C09199=1111.807,-65.980,-48.450,179.739,5.212,148.980
C09200=1111.812,-66.230,-48.440,179.738,5.207,148.979
C09201=1111.817,-66.480,-48.428,179.738,5.202,148.978
C09202=1111.823,-66.729,-48.417,179.737,5.197,148.977
C09203=1111.828,-66.979,-48.406,179.738,5.192,148.976
C09204=1111.833,-67.229,-48.395,179.737,5.187,148.975
C09205=1111.838,-67.478,-48.384,179.737,5.181,148.974
C09206=1111.843,-67.728,-48.373,179.737,5.176,148.972
C09207=1111.849,-67.978,-48.361,179.736,5.171,148.971
C09208=1111.854,-68.227,-48.350,179.737,5.166,148.970
C09209=1111.859,-68.477,-48.340,179.737,5.161,148.969
C09210=1111.864,-68.727,-48.328,179.736,5.155,148.968
C09211=1111.870,-68.976,-48.317,179.736,5.150,148.967
C09212=1111.875,-69.226,-48.306,179.736,5.145,148.966
C09213=1111.880,-69.475,-48.295,179.736,5.140,148.965
C09214=1111.885,-69.725,-48.285,179.736,5.135,148.964
C09215=1111.891,-69.975,-48.273,179.736,5.130,148.963
C09216=1111.896,-70.225,-48.263,179.735,5.124,148.962
C09217=1111.901,-70.475,-48.251,179.735,5.119,148.961
C09218=1111.906,-70.724,-48.240,179.735,5.114,148.959
C09219=1111.912,-70.974,-48.229,179.735,5.109,148.958
C09220=1111.917,-71.224,-48.218,179.735,5.104,148.957
C09221=1111.922,-71.473,-48.208,179.735,5.099,148.956
C09222=1111.927,-71.723,-48.197,179.735,5.094,148.955
C09223=1111.932,-71.972,-48.186,179.735,5.089,148.954
C09224=1111.937,-72.187,-48.176,179.735,5.084,148.953
C09225=1111.941,-72.403,-48.167,179.735,5.079,148.952
C09226=1111.946,-72.617,-48.157,179.735,5.075,148.951
C09227=1111.950,-72.832,-48.149,179.735,5.070,148.950
C09228=1111.955,-73.046,-48.139,179.735,5.066,148.949
C09229=1111.960,-73.262,-48.130,179.735,5.061,148.948
C09230=1111.963,-73.476,-48.120,179.735,5.057,148.947
C09231=1111.969,-73.691,-48.111,179.735,5.053,148.946
C09232=1111.973,-73.941,-48.100,179.735,5.048,148.945
C09233=1111.979,-74.190,-48.090,179.735,5.042,148.944
C09234=1111.984,-74.440,-48.079,179.735,5.037,148.943
C09235=1111.990,-74.690,-48.068,179.735,5.032,148.941
C09236=1111.995,-74.940,-48.057,179.736,5.027,148.940
C09237=1112.000,-75.189,-48.046,179.735,5.022,148.939
C09238=1112.005,-75.439,-48.036,179.735,5.017,148.938
C09239=1112.011,-75.689,-48.026,179.735,5.012,148.937
C09240=1112.016,-75.938,-48.014,179.736,5.007,148.936
C09241=1112.021,-76.188,-48.004,179.736,5.002,148.935
C09242=1112.026,-76.438,-47.993,179.735,4.996,148.933
C09243=1112.031,-76.687,-47.983,179.735,4.990,148.932
C09244=1112.037,-76.937,-47.971,179.736,4.985,148.931
C09245=1112.043,-77.187,-47.961,179.736,4.980,148.930
C09246=1112.048,-77.437,-47.950,179.736,4.975,148.929
C09247=1112.053,-77.686,-47.940,179.736,4.970,148.928
C09248=1112.058,-77.936,-47.929,179.736,4.965,148.926
C09249=1112.064,-78.186,-47.919,179.736,4.960,148.925
C09250=1112.068,-78.436,-47.908,179.737,4.954,148.924
C09251=1112.074,-78.685,-47.897,179.737,4.949,148.923
C09252=1112.079,-78.935,-47.887,179.737,4.944,148.922
C09253=1112.085,-79.185,-47.877,179.737,4.939,148.921
C09254=1112.089,-79.435,-47.865,179.737,4.934,148.919
C09255=1112.095,-79.684,-47.855,179.737,4.929,148.918
C09256=1112.100,-79.934,-47.845,179.738,4.924,148.917
C09257=1112.105,-80.184,-47.834,179.738,4.918,148.916
C09258=1112.111,-80.433,-47.823,179.738,4.914,148.915
C09259=1112.116,-80.683,-47.813,179.739,4.909,148.914
C09260=1112.121,-80.933,-47.803,179.739,4.903,148.912
C09261=1112.126,-81.183,-47.792,179.739,4.898,148.911
C09262=1112.132,-81.432,-47.782,179.740,4.893,148.910
C09263=1112.137,-81.683,-47.771,179.740,4.888,148.909
C09264=1112.142,-81.932,-47.760,179.740,4.883,148.907
C09265=1112.148,-82.181,-47.750,179.740,4.878,148.906
C09266=1112.153,-82.431,-47.740,179.740,4.873,148.905
C09267=1112.158,-82.681,-47.729,179.740,4.867,148.904
C09268=1112.163,-82.931,-47.719,179.741,4.862,148.903
C09269=1112.169,-83.181,-47.709,179.741,4.857,148.902
C09270=1112.174,-83.430,-47.699,179.742,4.853,148.900
C09271=1112.179,-83.680,-47.688,179.742,4.847,148.899
C09272=1112.184,-83.929,-47.677,179.742,4.842,148.898
C09273=1112.189,-84.179,-47.667,179.743,4.837,148.897
C09274=1112.195,-84.429,-47.657,179.743,4.832,148.895
C09275=1112.200,-84.678,-47.646,179.743,4.827,148.894
C09276=1112.205,-84.929,-47.636,179.744,4.822,148.893
C09277=1112.211,-85.178,-47.626,179.744,4.817,148.892
C09278=1112.216,-85.428,-47.615,179.744,4.812,148.891
C09279=1112.221,-85.678,-47.605,179.745,4.806,148.889
C09280=1112.226,-85.892,-47.597,179.745,4.802,148.888
C09281=1112.230,-86.108,-47.588,179.745,4.799,148.887
C09282=1112.235,-86.322,-47.579,179.745,4.793,148.886
C09283=1112.239,-86.538,-47.570,179.746,4.789,148.885
C09284=1112.244,-86.752,-47.561,179.746,4.785,148.884
C09285=1112.248,-86.967,-47.552,179.747,4.781,148.883
C09286=1112.253,-87.182,-47.543,179.746,4.776,148.882
C09287=1112.257,-87.397,-47.534,179.747,4.772,148.881
C09288=1112.263,-87.646,-47.524,179.747,4.767,148.880
C09289=1112.268,-87.896,-47.514,179.748,4.763,148.879
C09290=1112.273,-88.146,-47.504,179.748,4.757,148.877
C09291=1112.278,-88.395,-47.494,179.748,4.752,148.876
C09292=1112.284,-88.645,-47.483,179.749,4.747,148.875
C09293=1112.289,-88.896,-47.474,179.750,4.742,148.874
C09294=1112.295,-89.145,-47.463,179.750,4.737,148.872
C09295=1112.300,-89.395,-47.454,179.750,4.732,148.871
C09296=1112.305,-89.644,-47.444,179.751,4.728,148.870
C09297=1112.310,-89.894,-47.433,179.751,4.723,148.869
C09298=1112.316,-90.144,-47.423,179.751,4.717,148.868
C09299=1112.321,-90.393,-47.413,179.753,4.713,148.866
C09300=1112.326,-90.643,-47.403,179.753,4.707,148.865
C09301=1112.331,-90.893,-47.392,179.753,4.702,148.864
C09302=1112.337,-91.143,-47.382,179.754,4.698,148.863
C09303=1112.341,-91.392,-47.372,179.754,4.693,148.862
C09304=1112.347,-91.643,-47.363,179.754,4.688,148.860
C09305=1112.353,-91.892,-47.353,179.755,4.683,148.859
C09306=1112.358,-92.142,-47.342,179.755,4.678,148.858
C09307=1112.362,-92.392,-47.332,179.757,4.673,148.857
C09308=1112.368,-92.641,-47.322,179.757,4.668,148.855
C09309=1112.374,-92.891,-47.312,179.758,4.664,148.854
C09310=1112.380,-93.141,-47.302,179.758,4.659,148.853
C09311=1112.384,-93.391,-47.292,179.758,4.654,148.852
C09312=1112.389,-93.640,-47.282,179.759,4.649,148.851
C09313=1112.395,-93.890,-47.272,179.759,4.644,148.849
C09314=1112.400,-94.139,-47.262,179.760,4.640,148.848
C09315=1112.405,-94.390,-47.253,179.760,4.635,148.847
C09316=1112.411,-94.640,-47.242,179.760,4.630,148.846
C09317=1112.416,-94.889,-47.233,179.761,4.625,148.845
C09318=1112.421,-95.138,-47.223,179.761,4.620,148.843
C09319=1112.426,-95.389,-47.212,179.761,4.615,148.842
C09320=1112.431,-95.638,-47.203,179.762,4.611,148.841
C09321=1112.437,-95.888,-47.193,179.762,4.605,148.840
C09322=1112.443,-96.138,-47.183,179.763,4.600,148.839
C09323=1112.448,-96.387,-47.174,179.763,4.595,148.838
C09324=1112.453,-96.638,-47.163,179.764,4.591,148.836
C09325=1112.458,-96.887,-47.153,179.764,4.586,148.835
C09326=1112.463,-97.136,-47.143,179.764,4.580,148.834
C09327=1112.469,-97.387,-47.134,179.765,4.576,148.833
C09328=1112.475,-97.636,-47.124,179.765,4.571,148.832
C09329=1112.479,-97.886,-47.114,179.765,4.566,148.830
C09330=1112.485,-98.136,-47.104,179.765,4.561,148.829
C09331=1112.490,-98.385,-47.095,179.766,4.556,148.828
C09332=1112.495,-98.635,-47.084,179.766,4.551,148.827
C09333=1112.501,-98.885,-47.075,179.767,4.546,148.826
C09334=1112.506,-99.134,-47.065,179.767,4.541,148.824
C09335=1112.511,-99.385,-47.055,179.768,4.536,148.823
C09336=1112.516,-99.600,-47.047,179.767,4.532,148.822
C09337=1112.520,-99.814,-47.039,179.768,4.528,148.821
C09338=1112.524,-100.029,-47.030,179.769,4.523,148.820
C09339=1112.530,-100.245,-47.022,179.769,4.519,148.819
C09340=1112.534,-100.459,-47.013,179.769,4.515,148.818
C09341=1112.538,-100.674,-47.005,179.769,4.510,148.817
C09342=1112.543,-100.889,-46.996,179.770,4.506,148.816
C09343=1112.548,-101.104,-46.988,179.770,4.502,148.815
C09344=1112.553,-101.353,-46.979,179.770,4.497,148.814
C09345=1112.559,-101.604,-46.969,179.770,4.492,148.813
C09346=1112.563,-101.854,-46.959,179.771,4.487,148.812
C09347=1112.569,-102.103,-46.949,179.771,4.483,148.810
C09348=1112.574,-102.353,-46.940,179.772,4.477,148.809
C09349=1112.580,-102.603,-46.930,179.772,4.472,148.808
C09350=1112.585,-102.852,-46.921,179.772,4.467,148.807
C09351=1112.590,-103.102,-46.911,179.772,4.462,148.806
C09352=1112.596,-103.352,-46.902,179.773,4.458,148.804
C09353=1112.601,-103.601,-46.892,179.773,4.452,148.803
C09354=1112.606,-103.852,-46.882,179.774,4.447,148.802
C09355=1112.611,-104.101,-46.872,179.774,4.442,148.801
C09356=1112.617,-104.336,-46.864,179.775,4.438,148.800
C09357=1112.621,-104.571,-46.854,179.774,4.433,148.799
C09358=1112.626,-104.806,-46.846,179.775,4.428,148.797
C09359=1112.631,-105.041,-46.837,179.775,4.423,148.796
C09360=1112.637,-105.276,-46.828,179.776,4.418,148.795
C09361=1112.641,-105.511,-46.818,179.776,4.414,148.794
C09362=1112.646,-105.746,-46.810,179.776,4.409,148.793
C09363=1112.651,-105.980,-46.801,179.776,4.404,148.792
C09364=1112.656,-106.230,-46.792,179.777,4.400,148.790
C09365=1112.662,-106.480,-46.782,179.777,4.395,148.789
C09366=1112.667,-106.730,-46.773,179.778,4.389,148.788
C09367=1112.673,-106.980,-46.763,179.778,4.384,148.787
C09368=1112.678,-107.229,-46.754,179.778,4.379,148.786
C09369=1112.683,-107.479,-46.744,179.778,4.374,148.784
C09370=1112.689,-107.729,-46.735,179.779,4.370,148.783
C09371=1112.693,-107.978,-46.726,179.780,4.364,148.782
C09372=1112.699,-108.228,-46.716,179.780,4.359,148.781
C09373=1112.704,-108.478,-46.706,179.780,4.354,148.780
C09374=1112.709,-108.728,-46.698,179.780,4.349,148.778
C09375=1112.715,-108.978,-46.688,179.781,4.344,148.777
C09376=1112.720,-109.227,-46.678,179.781,4.339,148.776
C09377=1112.726,-109.477,-46.669,179.782,4.334,148.775
C09378=1112.731,-109.727,-46.660,179.782,4.329,148.774
C09379=1112.736,-109.976,-46.650,179.782,4.324,148.772
C09380=1112.742,-110.226,-46.641,179.782,4.319,148.771
C09381=1112.747,-110.476,-46.632,179.783,4.313,148.770
C09382=1112.752,-110.725,-46.622,179.783,4.308,148.769
C09383=1112.758,-110.976,-46.613,179.784,4.303,148.767
C09384=1112.763,-111.225,-46.604,179.784,4.298,148.766
C09385=1112.768,-111.475,-46.595,179.784,4.293,148.765
C09386=1112.774,-111.725,-46.585,179.785,4.288,148.764
C09387=1112.779,-111.975,-46.576,179.785,4.283,148.763
C09388=1112.784,-112.225,-46.567,179.785,4.278,148.761
C09389=1112.789,-112.474,-46.558,179.786,4.273,148.760
C09390=1112.795,-112.724,-46.548,179.786,4.268,148.759
C09391=1112.800,-112.974,-46.539,179.786,4.262,148.758
C09392=1112.805,-113.204,-46.531,179.787,4.257,148.757
C09393=1112.810,-113.434,-46.523,179.787,4.253,148.755
C09394=1112.815,-113.663,-46.514,179.788,4.248,148.754
C09395=1112.820,-113.893,-46.505,179.787,4.243,148.753
C09396=1112.825,-114.124,-46.497,179.788,4.239,148.752
C09397=1112.829,-114.354,-46.489,179.788,4.233,148.751
C09398=1112.834,-114.584,-46.480,179.789,4.229,148.750
C09399=1112.840,-114.813,-46.472,179.789,4.224,148.749
C09400=1112.845,-115.063,-46.463,179.789,4.219,148.747
C09401=1112.850,-115.313,-46.454,179.790,4.214,148.746
C09402=1112.856,-115.563,-46.444,179.790,4.208,148.745
C09403=1112.861,-115.812,-46.435,179.791,4.203,148.743
C09404=1112.866,-116.062,-46.426,179.791,4.198,148.742
C09405=1112.871,-116.312,-46.417,179.791,4.193,148.741
C09406=1112.876,-116.562,-46.408,179.791,4.188,148.740
C09407=1112.882,-116.812,-46.399,179.792,4.183,148.739
C09408=1112.888,-117.061,-46.390,179.792,4.177,148.737
C09409=1112.893,-117.311,-46.381,179.793,4.172,148.736
C09410=1112.898,-117.561,-46.372,179.793,4.167,148.735
C09411=1112.903,-117.810,-46.363,179.793,4.162,148.734
C09412=1112.909,-118.061,-46.354,179.794,4.156,148.732
C09413=1112.915,-118.310,-46.345,179.794,4.151,148.731
C09414=1112.919,-118.560,-46.335,179.795,4.146,148.730
C09415=1112.925,-118.810,-46.327,179.795,4.141,148.728
C09416=1112.930,-119.059,-46.318,179.795,4.135,148.727
C09417=1112.935,-119.309,-46.309,179.796,4.130,148.726
C09418=1112.941,-119.558,-46.300,179.796,4.125,148.725
C09419=1112.947,-119.809,-46.291,179.797,4.119,148.723
C09420=1112.952,-120.058,-46.282,179.797,4.114,148.722
C09421=1112.957,-120.308,-46.273,179.797,4.109,148.721
C09422=1112.962,-120.558,-46.264,179.797,4.104,148.720
C09423=1112.968,-120.807,-46.255,179.798,4.098,148.718
C09424=1112.973,-121.057,-46.247,179.799,4.093,148.717
C09425=1112.978,-121.307,-46.238,179.799,4.088,148.716
C09426=1112.984,-121.557,-46.229,179.799,4.083,148.715
C09427=1112.989,-121.807,-46.221,179.800,4.077,148.713
C09428=1112.994,-122.057,-46.212,179.800,4.072,148.712
C09429=1113.000,-122.306,-46.203,179.800,4.066,148.711
C09430=1113.006,-122.556,-46.194,179.800,4.061,148.710
C09431=1113.011,-122.806,-46.185,179.801,4.056,148.708
C09432=1113.016,-123.056,-46.176,179.801,4.050,148.707
C09433=1113.021,-123.306,-46.167,179.802,4.045,148.706
C09434=1113.027,-123.555,-46.158,179.802,4.040,148.704
C09435=1113.032,-123.805,-46.150,179.803,4.034,148.703
C09436=1113.037,-124.055,-46.141,179.803,4.029,148.702
C09437=1113.043,-124.305,-46.132,179.804,4.024,148.700
C09438=1113.048,-124.555,-46.124,179.804,4.019,148.699
C09439=1113.054,-124.804,-46.115,179.804,4.013,148.698
C09440=1113.059,-125.054,-46.106,179.805,4.007,148.696
C09441=1113.064,-125.304,-46.097,179.805,4.002,148.695
C09442=1113.069,-125.554,-46.088,179.805,3.997,148.694
C09443=1113.075,-125.804,-46.081,179.806,3.991,148.692
C09444=1113.080,-126.054,-46.072,179.806,3.986,148.691
C09445=1113.086,-126.303,-46.063,179.807,3.981,148.690
C09446=1113.091,-126.553,-46.054,179.807,3.974,148.689
C09447=1113.096,-126.802,-46.045,179.807,3.969,148.687
C09448=1113.101,-127.018,-46.039,179.808,3.965,148.686
C09449=1113.105,-127.234,-46.031,179.808,3.960,148.685
C09450=1113.110,-127.449,-46.023,179.808,3.955,148.684
C09451=1113.115,-127.664,-46.016,179.809,3.951,148.683
C09452=1113.119,-127.879,-46.009,179.809,3.946,148.682
C09453=1113.124,-128.094,-46.001,179.810,3.942,148.681
C09454=1113.128,-128.309,-45.994,179.810,3.936,148.679
C09455=1113.132,-128.523,-45.987,179.810,3.932,148.678
C09456=1112.710,-128.514,-46.013,179.818,3.936,148.677
C09457=1112.703,-128.193,-46.024,179.817,3.943,148.679
C09458=1112.697,-127.871,-46.035,179.817,3.950,148.680
C09459=1112.690,-127.549,-46.046,179.816,3.957,148.682
C09460=1112.683,-127.227,-46.057,179.816,3.964,148.684
C09461=1112.677,-126.978,-46.065,179.815,3.970,148.685
C09462=1112.671,-126.728,-46.074,179.814,3.975,148.686
C09463=1112.666,-126.478,-46.083,179.814,3.980,148.688
C09464=1112.661,-126.228,-46.092,179.813,3.986,148.689
C09465=1112.655,-125.979,-46.100,179.813,3.991,148.690
C09466=1112.650,-125.728,-46.109,179.813,3.997,148.691
C09467=1112.645,-125.479,-46.118,179.812,4.003,148.693
C09468=1112.639,-125.229,-46.126,179.812,4.008,148.694
C09469=1112.634,-124.980,-46.135,179.811,4.013,148.696
C09470=1112.629,-124.730,-46.144,179.811,4.018,148.697
C09471=1112.623,-124.480,-46.153,179.811,4.024,148.698
C09472=1112.618,-124.230,-46.162,179.810,4.029,148.700
C09473=1112.613,-123.980,-46.171,179.810,4.034,148.701
C09474=1112.607,-123.730,-46.178,179.810,4.040,148.702
C09475=1112.602,-123.481,-46.187,179.809,4.046,148.703
C09476=1112.597,-123.231,-46.196,179.809,4.051,148.705
C09477=1112.591,-122.981,-46.205,179.809,4.056,148.706
C09478=1112.586,-122.731,-46.214,179.808,4.061,148.707
C09479=1112.581,-122.481,-46.223,179.807,4.067,148.709
C09480=1112.575,-122.232,-46.231,179.807,4.072,148.710
C09481=1112.570,-121.982,-46.240,179.807,4.077,148.711
C09482=1112.565,-121.732,-46.249,179.806,4.083,148.712
C09483=1112.560,-121.482,-46.258,179.806,4.088,148.714
C09484=1112.554,-121.232,-46.268,179.805,4.093,148.715
C09485=1112.549,-120.982,-46.277,179.805,4.098,148.716
C09486=1112.543,-120.733,-46.285,179.804,4.104,148.718
C09487=1112.538,-120.483,-46.294,179.804,4.109,148.719
C09488=1112.533,-120.234,-46.303,179.804,4.114,148.720
C09489=1112.527,-119.984,-46.312,179.804,4.119,148.721
C09490=1112.522,-119.734,-46.321,179.803,4.126,148.723
C09491=1112.517,-119.484,-46.330,179.803,4.131,148.724
C09492=1112.511,-119.234,-46.339,179.803,4.136,148.725
C09493=1112.505,-118.985,-46.348,179.802,4.141,148.726
C09494=1112.500,-118.735,-46.356,179.802,4.146,148.727
C09495=1112.495,-118.485,-46.365,179.801,4.152,148.729
C09496=1112.490,-118.235,-46.374,179.801,4.157,148.730
C09497=1112.485,-117.985,-46.383,179.801,4.162,148.731
C09498=1112.479,-117.735,-46.393,179.801,4.167,148.733
C09499=1112.474,-117.486,-46.402,179.800,4.173,148.734
C09500=1112.469,-117.236,-46.411,179.800,4.178,148.735
C09501=1112.464,-116.986,-46.420,179.799,4.183,148.736
C09502=1112.458,-116.737,-46.429,179.799,4.188,148.738
C09503=1112.452,-116.487,-46.438,179.799,4.194,148.739
C09504=1112.447,-116.237,-46.447,179.798,4.198,148.740
C09505=1112.442,-115.987,-46.456,179.798,4.203,148.741
C09506=1112.437,-115.737,-46.465,179.797,4.209,148.743
C09507=1112.431,-115.488,-46.475,179.797,4.214,148.744
C09508=1112.426,-115.238,-46.484,179.796,4.219,148.745
C09509=1112.421,-115.020,-46.492,179.797,4.224,148.746
C09510=1112.417,-114.804,-46.499,179.796,4.228,148.747
C09511=1112.412,-114.589,-46.507,179.796,4.233,148.748
C09512=1112.408,-114.374,-46.516,179.795,4.237,148.749
C09513=1112.403,-114.159,-46.523,179.795,4.241,148.750
C09514=1112.398,-113.944,-46.531,179.795,4.246,148.751
C09515=1112.394,-113.729,-46.539,179.794,4.250,148.753
C09516=1112.389,-113.514,-46.547,179.794,4.255,148.754
C09517=1112.384,-113.299,-46.554,179.794,4.259,148.755
C09518=1112.380,-113.084,-46.563,179.793,4.263,148.756
C09519=1112.375,-112.834,-46.572,179.793,4.269,148.757
C09520=1112.369,-112.584,-46.582,179.793,4.274,148.758
C09521=1112.364,-112.334,-46.590,179.792,4.279,148.759
C09522=1112.359,-112.085,-46.600,179.792,4.284,148.761
C09523=1112.353,-111.834,-46.610,179.791,4.290,148.762
C09524=1112.348,-111.585,-46.618,179.791,4.295,148.763
C09525=1112.343,-111.335,-46.628,179.791,4.300,148.764
C09526=1112.337,-111.085,-46.638,179.791,4.305,148.766
C09527=1112.332,-110.835,-46.646,179.790,4.309,148.767
C09528=1112.327,-110.586,-46.656,179.790,4.315,148.768
C09529=1112.321,-110.336,-46.666,179.789,4.320,148.769
C09530=1112.316,-110.086,-46.674,179.789,4.325,148.770
C09531=1112.311,-109.837,-46.684,179.789,4.330,148.772
C09532=1112.305,-109.587,-46.694,179.789,4.335,148.773
C09533=1112.300,-109.337,-46.702,179.788,4.340,148.774
C09534=1112.295,-109.087,-46.713,179.788,4.346,148.775
C09535=1112.289,-108.837,-46.722,179.787,4.350,148.776
C09536=1112.284,-108.588,-46.730,179.787,4.355,148.778
C09537=1112.279,-108.338,-46.741,179.786,4.361,148.779
C09538=1112.274,-108.088,-46.750,179.786,4.366,148.780
C09539=1112.268,-107.839,-46.760,179.786,4.371,148.782
C09540=1112.263,-107.589,-46.769,179.786,4.376,148.783
C09541=1112.258,-107.339,-46.778,179.785,4.381,148.784
C09542=1112.252,-107.089,-46.788,179.784,4.386,148.785
C09543=1112.247,-106.840,-46.797,179.784,4.391,148.786
C09544=1112.241,-106.590,-46.807,179.784,4.396,148.788
C09545=1112.236,-106.340,-46.816,179.784,4.401,148.789
C09546=1112.231,-106.091,-46.825,179.784,4.406,148.790
C09547=1112.226,-105.840,-46.835,179.783,4.411,148.791
C09548=1112.221,-105.590,-46.844,179.782,4.416,148.792
C09549=1112.215,-105.341,-46.854,179.782,4.421,148.794
C09550=1112.210,-105.091,-46.863,179.782,4.426,148.795
C09551=1112.204,-104.841,-46.873,179.782,4.431,148.796
C09552=1112.199,-104.591,-46.882,179.782,4.436,148.797
C09553=1112.194,-104.342,-46.893,179.781,4.441,148.798
C09554=1112.188,-104.092,-46.901,179.780,4.446,148.800
C09555=1112.183,-103.843,-46.912,179.780,4.451,148.801
C09556=1112.178,-103.593,-46.921,179.780,4.456,148.802
C09557=1112.173,-103.342,-46.931,179.780,4.461,148.803
C09558=1112.168,-103.093,-46.941,179.779,4.466,148.804
C09559=1112.162,-102.843,-46.950,179.779,4.471,148.806
C09560=1112.157,-102.594,-46.960,179.778,4.476,148.807
C09561=1112.151,-102.344,-46.969,179.778,4.481,148.808
C09562=1112.146,-102.094,-46.979,179.778,4.486,148.809
C09563=1112.140,-101.844,-46.988,179.777,4.491,148.810
C09564=1112.136,-101.594,-46.998,179.777,4.496,148.812
C09565=1112.131,-101.345,-47.009,179.777,4.501,148.813
C09566=1112.125,-101.095,-47.018,179.777,4.506,148.814
C09567=1112.120,-100.880,-47.026,179.776,4.510,148.815
C09568=1112.116,-100.666,-47.035,179.775,4.514,148.816
C09569=1112.111,-100.450,-47.043,179.775,4.518,148.817
C09570=1112.107,-100.235,-47.051,179.775,4.523,148.818
C09571=1112.102,-100.021,-47.060,179.775,4.527,148.819
C09572=1112.098,-99.805,-47.069,179.774,4.531,148.820
C09573=1112.093,-99.590,-47.076,179.774,4.535,148.821
C09574=1112.088,-99.376,-47.085,179.774,4.540,148.822
C09575=1112.083,-99.126,-47.095,179.774,4.545,148.823
C09576=1112.079,-98.876,-47.105,179.773,4.550,148.824
C09577=1112.073,-98.626,-47.114,179.773,4.555,148.826
C09578=1112.067,-98.377,-47.125,179.773,4.560,148.827
C09579=1112.062,-98.127,-47.134,179.772,4.564,148.828
C09580=1112.057,-97.877,-47.144,179.772,4.570,148.829
C09581=1112.051,-97.627,-47.154,179.772,4.575,148.830
C09582=1112.046,-97.378,-47.164,179.771,4.579,148.832
C09583=1112.041,-97.128,-47.173,179.771,4.584,148.833
C09584=1112.035,-96.878,-47.184,179.770,4.589,148.834
C09585=1112.031,-96.628,-47.194,179.770,4.594,148.835
C09586=1112.025,-96.379,-47.204,179.769,4.599,148.836
C09587=1112.019,-96.128,-47.213,179.769,4.604,148.838
C09588=1112.014,-95.879,-47.223,179.769,4.609,148.839
C09589=1112.009,-95.630,-47.233,179.769,4.614,148.840
C09590=1112.004,-95.379,-47.244,179.768,4.619,148.841
C09591=1111.999,-95.130,-47.253,179.768,4.624,148.842
C09592=1111.993,-94.880,-47.263,179.768,4.629,148.843
C09593=1111.987,-94.631,-47.273,179.767,4.633,148.845
C09594=1111.983,-94.381,-47.283,179.767,4.638,148.846
C09595=1111.978,-94.131,-47.293,179.766,4.644,148.847
C09596=1111.972,-93.882,-47.303,179.766,4.648,148.848
C09597=1111.967,-93.632,-47.312,179.765,4.653,148.849
C09598=1111.962,-93.381,-47.323,179.765,4.657,148.851
C09599=1111.956,-93.132,-47.333,179.764,4.663,148.852
C09600=1111.951,-92.882,-47.343,179.764,4.667,148.853
C09601=1111.946,-92.632,-47.353,179.763,4.672,148.854
C09602=1111.941,-92.383,-47.363,179.763,4.678,148.856
C09603=1111.935,-92.133,-47.373,179.762,4.682,148.857
C09604=1111.929,-91.883,-47.383,179.762,4.687,148.858
C09605=1111.925,-91.633,-47.393,179.761,4.691,148.859
C09606=1111.919,-91.384,-47.403,179.761,4.697,148.860
C09607=1111.914,-91.134,-47.414,179.761,4.702,148.862
C09608=1111.909,-90.884,-47.424,179.760,4.706,148.863
C09609=1111.904,-90.635,-47.434,179.760,4.711,148.864
C09610=1111.898,-90.385,-47.444,179.759,4.717,148.865
C09611=1111.893,-90.136,-47.454,179.758,4.721,148.867
C09612=1111.888,-89.885,-47.465,179.758,4.726,148.868
C09613=1111.882,-89.636,-47.475,179.758,4.731,148.869
C09614=1111.877,-89.387,-47.485,179.757,4.736,148.870
C09615=1111.872,-89.136,-47.494,179.757,4.741,148.871
C09616=1111.866,-88.886,-47.505,179.757,4.746,148.872
C09617=1111.861,-88.637,-47.515,179.755,4.751,148.874
C09618=1111.856,-88.386,-47.525,179.755,4.756,148.875
C09619=1111.851,-88.137,-47.535,179.755,4.761,148.876
C09620=1111.845,-87.888,-47.545,179.755,4.766,148.877
C09621=1111.840,-87.637,-47.556,179.754,4.771,148.879
C09622=1111.835,-87.388,-47.566,179.754,4.776,148.880
C09623=1111.831,-87.173,-47.575,179.753,4.780,148.881
C09624=1111.826,-86.958,-47.584,179.753,4.785,148.882
C09625=1111.821,-86.744,-47.593,179.753,4.789,148.883
C09626=1111.817,-86.528,-47.602,179.752,4.793,148.884
C09627=1111.812,-86.314,-47.610,179.752,4.797,148.885
C09628=1111.808,-86.099,-47.620,179.752,4.802,148.886
C09629=1111.803,-85.884,-47.628,179.752,4.806,148.887
C09630=1111.799,-85.669,-47.637,179.751,4.811,148.888
C09631=1111.794,-85.419,-47.647,179.751,4.816,148.889
C09632=1111.789,-85.169,-47.657,179.750,4.821,148.891
C09633=1111.783,-84.920,-47.668,179.750,4.826,148.892
C09634=1111.778,-84.671,-47.678,179.750,4.830,148.893
C09635=1111.773,-84.420,-47.689,179.749,4.836,148.894
C09636=1111.767,-84.171,-47.699,179.749,4.841,148.895
C09637=1111.761,-83.921,-47.709,179.749,4.846,148.897
C09638=1111.756,-83.671,-47.720,179.748,4.851,148.898
C09639=1111.751,-83.422,-47.730,179.748,4.856,148.899
C09640=1111.746,-83.171,-47.741,179.748,4.862,148.900
C09641=1111.741,-82.922,-47.750,179.747,4.866,148.901
C09642=1111.736,-82.672,-47.762,179.747,4.871,148.903
C09643=1111.731,-82.423,-47.772,179.747,4.876,148.904
C09644=1111.725,-82.173,-47.782,179.747,4.881,148.905
C09645=1111.720,-81.923,-47.793,179.747,4.887,148.906
C09646=1111.715,-81.674,-47.803,179.746,4.892,148.907
C09647=1111.710,-81.424,-47.814,179.746,4.897,148.909
C09648=1111.704,-81.174,-47.824,179.746,4.902,148.910
C09649=1111.699,-80.924,-47.835,179.745,4.908,148.911
C09650=1111.694,-80.675,-47.845,179.745,4.913,148.912
C09651=1111.688,-80.425,-47.855,179.745,4.918,148.913
C09652=1111.683,-80.175,-47.867,179.745,4.923,148.915
C09653=1111.678,-79.926,-47.877,179.745,4.928,148.916
C09654=1111.673,-79.676,-47.888,179.745,4.933,148.917
C09655=1111.667,-79.426,-47.898,179.744,4.938,148.918
C09656=1111.662,-79.176,-47.909,179.744,4.943,148.919
C09657=1111.657,-78.927,-47.919,179.744,4.948,148.921
C09658=1111.652,-78.677,-47.930,179.743,4.953,148.922
C09659=1111.646,-78.427,-47.940,179.743,4.958,148.923
C09660=1111.641,-78.177,-47.952,179.743,4.963,148.924
C09661=1111.635,-77.928,-47.962,179.743,4.968,148.925
C09662=1111.630,-77.677,-47.973,179.743,4.974,148.926
C09663=1111.625,-77.428,-47.984,179.743,4.979,148.928
C09664=1111.620,-77.178,-47.994,179.742,4.984,148.929
C09665=1111.614,-76.929,-48.004,179.743,4.990,148.930
C09666=1111.610,-76.679,-48.016,179.743,4.995,148.931
C09667=1111.604,-76.430,-48.026,179.743,5.000,148.932
C09668=1111.599,-76.179,-48.036,179.742,5.005,148.933
C09669=1111.594,-75.930,-48.047,179.742,5.010,148.935
C09670=1111.589,-75.680,-48.058,179.742,5.016,148.936
C09671=1111.582,-75.430,-48.069,179.742,5.021,148.937
C09672=1111.578,-75.181,-48.080,179.742,5.026,148.938
C09673=1111.572,-74.931,-48.090,179.742,5.031,148.939
C09674=1111.567,-74.681,-48.102,179.742,5.036,148.940
C09675=1111.562,-74.432,-48.112,179.742,5.041,148.941
C09676=1111.557,-74.182,-48.123,179.742,5.046,148.943
C09677=1111.552,-73.933,-48.133,179.742,5.051,148.944
C09678=1111.546,-73.682,-48.144,179.741,5.056,148.945
C09679=1111.542,-73.468,-48.154,179.742,5.061,148.946
C09680=1111.537,-73.253,-48.163,179.742,5.065,148.947
C09681=1111.533,-73.038,-48.173,179.741,5.070,148.948
C09682=1111.528,-72.824,-48.182,179.741,5.074,148.949
C09683=1111.524,-72.609,-48.191,179.742,5.079,148.950
C09684=1111.519,-72.394,-48.201,179.741,5.083,148.951
C09685=1111.514,-72.179,-48.210,179.742,5.088,148.952
C09686=1111.511,-71.964,-48.219,179.742,5.092,148.953
C09687=1111.504,-71.715,-48.230,179.742,5.098,148.954
C09688=1111.500,-71.465,-48.242,179.742,5.103,148.955
C09689=1111.495,-71.215,-48.252,179.742,5.108,148.956
C09690=1111.489,-70.966,-48.263,179.741,5.113,148.957
C09691=1111.484,-70.716,-48.274,179.742,5.118,148.958
C09692=1111.478,-70.466,-48.285,179.742,5.123,148.959
C09693=1111.474,-70.217,-48.296,179.742,5.128,148.961
C09694=1111.469,-69.966,-48.307,179.742,5.134,148.962
C09695=1111.463,-69.717,-48.319,179.742,5.139,148.963
C09696=1111.458,-69.467,-48.329,179.742,5.144,148.964
C09697=1111.453,-69.217,-48.340,179.742,5.149,148.965
C09698=1111.448,-68.968,-48.351,179.743,5.154,148.966
C09699=1111.442,-68.718,-48.362,179.742,5.159,148.967
C09700=1111.437,-68.469,-48.373,179.743,5.165,148.968
C09701=1111.432,-68.219,-48.385,179.743,5.170,148.969
C09702=1111.426,-67.969,-48.396,179.743,5.175,148.970
C09703=1111.421,-67.720,-48.407,179.743,5.180,148.971
C09704=1111.416,-67.470,-48.418,179.743,5.185,148.972
C09705=1111.410,-67.220,-48.429,179.743,5.190,148.974
C09706=1111.405,-66.971,-48.440,179.744,5.195,148.974
C09707=1111.400,-66.721,-48.451,179.744,5.200,148.976
C09708=1111.395,-66.471,-48.463,179.744,5.206,148.977
C09709=1111.390,-66.221,-48.474,179.744,5.210,148.978
C09710=1111.385,-65.972,-48.485,179.744,5.216,148.979
C09711=1111.379,-65.722,-48.497,179.745,5.221,148.980
C09712=1111.374,-65.472,-48.507,179.745,5.226,148.981
C09713=1111.369,-65.223,-48.518,179.745,5.231,148.982
C09714=1111.364,-64.973,-48.530,179.745,5.236,148.983
C09715=1111.359,-64.723,-48.541,179.746,5.241,148.984
C09716=1111.353,-64.473,-48.553,179.746,5.247,148.985
C09717=1111.348,-64.224,-48.563,179.747,5.252,148.986
C09718=1111.343,-63.974,-48.575,179.746,5.257,148.987
C09719=1111.338,-63.724,-48.587,179.747,5.261,148.988
C09720=1111.333,-63.475,-48.598,179.747,5.266,148.989
C09721=1111.327,-63.225,-48.609,179.748,5.272,148.990
C09722=1111.322,-62.975,-48.620,179.748,5.277,148.991
C09723=1111.317,-62.726,-48.631,179.748,5.282,148.992
C09724=1111.312,-62.476,-48.643,179.748,5.287,148.993
C09725=1111.307,-62.227,-48.654,179.749,5.292,148.994
C09726=1111.301,-61.977,-48.666,179.750,5.297,148.995
C09727=1111.296,-61.727,-48.677,179.750,5.302,148.996
C09728=1111.291,-61.477,-48.689,179.750,5.307,148.997
C09729=1111.286,-61.228,-48.700,179.751,5.313,148.998
C09730=1111.280,-60.978,-48.711,179.751,5.317,148.999
C09731=1111.275,-60.728,-48.723,179.751,5.322,149.000
C09732=1111.270,-60.478,-48.734,179.752,5.327,149.001
C09733=1111.265,-60.229,-48.746,179.752,5.332,149.002
C09734=1111.260,-59.979,-48.758,179.753,5.338,149.003
C09735=1111.255,-59.764,-48.767,179.753,5.341,149.004
C09736=1111.250,-59.550,-48.777,179.753,5.345,149.005
C09737=1111.246,-59.335,-48.787,179.752,5.349,149.006
C09738=1111.242,-59.120,-48.797,179.752,5.353,149.007
C09739=1111.237,-58.906,-48.807,179.752,5.357,149.008
C09740=1111.232,-58.691,-48.817,179.752,5.361,149.008
C09741=1111.228,-58.476,-48.827,179.752,5.366,149.009
C09742=1111.224,-58.261,-48.837,179.752,5.370,149.010
C09743=1111.219,-58.011,-48.848,179.752,5.374,149.011
C09744=1111.213,-57.762,-48.860,179.752,5.379,149.012
C09745=1111.209,-57.513,-48.872,179.752,5.384,149.014
C09746=1111.203,-57.263,-48.884,179.751,5.388,149.014
C09747=1111.198,-57.013,-48.896,179.751,5.393,149.016
C09748=1111.193,-56.764,-48.907,179.751,5.398,149.017
C09749=1111.188,-56.514,-48.919,179.751,5.402,149.018
C09750=1111.183,-56.264,-48.930,179.751,5.407,149.019
C09751=1111.178,-56.014,-48.942,179.751,5.411,149.020
C09752=1111.172,-55.765,-48.953,179.751,5.416,149.021
C09753=1111.167,-55.515,-48.965,179.751,5.422,149.022
C09754=1111.161,-55.265,-48.977,179.750,5.426,149.023
C09755=1111.157,-55.016,-48.988,179.750,5.431,149.024
C09756=1111.152,-54.767,-49.000,179.750,5.436,149.025
C09757=1111.146,-54.517,-49.012,179.750,5.440,149.026
C09758=1111.142,-54.267,-49.024,179.750,5.445,149.027
C09759=1111.136,-54.017,-49.036,179.749,5.449,149.029
C09760=1111.131,-53.767,-49.047,179.750,5.454,149.029
C09761=1111.126,-53.517,-49.059,179.750,5.459,149.031
C09762=1111.120,-53.268,-49.070,179.749,5.463,149.032
C09763=1111.115,-53.019,-49.083,179.749,5.468,149.033
C09764=1111.110,-52.769,-49.094,179.749,5.473,149.034
C09765=1111.105,-52.519,-49.106,179.749,5.478,149.035
C09766=1111.099,-52.269,-49.118,179.749,5.482,149.036
C09767=1111.095,-52.020,-49.129,179.748,5.487,149.037
C09768=1111.089,-51.770,-49.142,179.748,5.492,149.038
C09769=1111.084,-51.521,-49.154,179.749,5.497,149.039
C09770=1111.079,-51.271,-49.165,179.748,5.501,149.040
C09771=1111.074,-51.021,-49.177,179.748,5.506,149.041
C09772=1111.069,-50.772,-49.189,179.748,5.511,149.042
C09773=1111.063,-50.522,-49.201,179.748,5.515,149.044
C09774=1111.059,-50.272,-49.213,179.748,5.520,149.045
C09775=1111.053,-50.022,-49.225,179.747,5.524,149.046
C09776=1111.048,-49.773,-49.237,179.747,5.529,149.047
C09777=1111.043,-49.523,-49.249,179.747,5.534,149.048
C09778=1111.038,-49.273,-49.260,179.747,5.538,149.049
C09779=1111.032,-49.024,-49.272,179.747,5.544,149.050
C09780=1111.027,-48.775,-49.284,179.747,5.549,149.051
C09781=1111.021,-48.525,-49.296,179.747,5.553,149.052
C09782=1111.016,-48.275,-49.308,179.747,5.558,149.053
C09783=1111.012,-48.026,-49.320,179.746,5.562,149.054
C09784=1111.006,-47.776,-49.332,179.746,5.567,149.055
C09785=1111.001,-47.526,-49.344,179.746,5.572,149.056
C09786=1110.996,-47.277,-49.357,179.746,5.576,149.058
C09787=1110.991,-47.027,-49.368,179.746,5.581,149.059
C09788=1110.985,-46.777,-49.380,179.746,5.586,149.060
C09789=1110.980,-46.528,-49.392,179.745,5.590,149.061
C09790=1110.975,-46.278,-49.404,179.745,5.596,149.062
C09791=1110.971,-46.064,-49.415,179.745,5.600,149.063
C09792=1110.967,-45.849,-49.425,179.745,5.603,149.064
C09793=1110.961,-45.634,-49.436,179.745,5.607,149.065
C09794=1110.957,-45.419,-49.446,179.745,5.611,149.066
C09795=1110.953,-45.204,-49.456,179.744,5.615,149.066
C09796=1110.949,-44.990,-49.467,179.744,5.619,149.067
C09797=1110.944,-44.775,-49.478,179.745,5.624,149.068
C09798=1110.940,-44.561,-49.488,179.744,5.628,149.069
C09799=1110.935,-44.311,-49.500,179.744,5.632,149.070
C09800=1110.929,-44.061,-49.512,179.744,5.637,149.072
C09801=1110.925,-43.812,-49.524,179.743,5.642,149.073
C09802=1110.919,-43.562,-49.536,179.744,5.646,149.074
C09803=1110.914,-43.313,-49.549,179.743,5.652,149.075
C09804=1110.909,-43.063,-49.560,179.743,5.656,149.076
C09805=1110.904,-42.813,-49.573,179.743,5.661,149.077
C09806=1110.898,-42.563,-49.585,179.744,5.667,149.078
C09807=1110.893,-42.314,-49.598,179.744,5.671,149.079
C09808=1110.888,-42.064,-49.609,179.745,5.677,149.080
C09809=1110.883,-41.815,-49.622,179.746,5.682,149.081
C09810=1110.877,-41.565,-49.634,179.746,5.686,149.082
C09811=1110.872,-41.316,-49.647,179.747,5.692,149.082
C09812=1110.868,-41.065,-49.658,179.748,5.697,149.083
C09813=1110.863,-40.816,-49.671,179.748,5.701,149.084
C09814=1110.858,-40.567,-49.683,179.749,5.707,149.085
C09815=1110.852,-40.317,-49.695,179.750,5.712,149.086
C09816=1110.847,-40.067,-49.708,179.750,5.716,149.087
C09817=1110.842,-39.817,-49.720,179.750,5.721,149.088
C09818=1110.837,-39.568,-49.732,179.752,5.726,149.089
C09819=1110.831,-39.319,-49.745,179.752,5.731,149.090
C09820=1110.827,-39.068,-49.757,179.753,5.736,149.090
C09821=1110.821,-38.819,-49.770,179.753,5.741,149.091
C09822=1110.816,-38.570,-49.782,179.754,5.745,149.092
C09823=1110.811,-38.320,-49.794,179.754,5.750,149.093
C09824=1110.805,-38.070,-49.807,179.755,5.755,149.094
C09825=1110.800,-37.821,-49.820,179.755,5.759,149.095
C09826=1110.794,-37.571,-49.832,179.756,5.764,149.096
C09827=1110.790,-37.321,-49.845,179.756,5.769,149.097
C09828=1110.785,-37.071,-49.858,179.757,5.773,149.097
C09829=1110.780,-36.822,-49.870,179.757,5.778,149.098
C09830=1110.774,-36.572,-49.882,179.758,5.783,149.099
C09831=1110.769,-36.323,-49.895,179.759,5.787,149.100
C09832=1110.765,-36.073,-49.908,179.759,5.792,149.101
C09833=1110.759,-35.824,-49.920,179.760,5.797,149.102
C09834=1110.754,-35.574,-49.932,179.760,5.801,149.103
C09835=1110.749,-35.324,-49.945,179.761,5.806,149.104
C09836=1110.743,-35.075,-49.958,179.761,5.811,149.105
C09837=1110.739,-34.825,-49.971,179.761,5.814,149.105
C09838=1110.733,-34.575,-49.983,179.762,5.819,149.106
C09839=1110.728,-34.325,-49.995,179.762,5.824,149.107
C09840=1110.723,-34.076,-50.008,179.763,5.829,149.108
C09841=1110.718,-33.827,-50.021,179.763,5.833,149.109
C09842=1110.713,-33.577,-50.033,179.763,5.837,149.110
C09843=1110.707,-33.327,-50.047,179.763,5.842,149.111
C09844=1110.702,-33.078,-50.059,179.764,5.846,149.111
C09845=1110.697,-32.828,-50.071,179.764,5.850,149.112
C09846=1110.692,-32.578,-50.084,179.765,5.855,149.113
C09847=1110.688,-32.363,-50.095,179.765,5.859,149.114
C09848=1110.683,-32.149,-50.106,179.765,5.862,149.115
C09849=1110.679,-31.934,-50.117,179.765,5.866,149.115
C09850=1110.675,-31.720,-50.128,179.765,5.870,149.116
C09851=1110.670,-31.506,-50.140,179.766,5.874,149.117
C09852=1110.666,-31.291,-50.150,179.766,5.878,149.118
C09853=1110.661,-31.076,-50.161,179.766,5.882,149.119
C09854=1110.657,-30.862,-50.172,179.767,5.885,149.119
C09855=1110.652,-30.613,-50.184,179.766,5.889,149.120
C09856=1110.646,-30.362,-50.198,179.767,5.894,149.121
C09857=1110.641,-30.113,-50.210,179.766,5.898,149.122
C09858=1110.636,-29.864,-50.223,179.767,5.903,149.123
C09859=1110.632,-29.614,-50.236,179.767,5.907,149.124
C09860=1110.626,-29.364,-50.249,179.767,5.912,149.125
C09861=1110.621,-29.115,-50.262,179.767,5.916,149.126
C09862=1110.616,-28.865,-50.275,179.767,5.920,149.127
C09863=1110.611,-28.615,-50.287,179.767,5.924,149.128
C09864=1110.605,-28.366,-50.300,179.767,5.929,149.129
C09865=1110.601,-28.116,-50.313,179.767,5.933,149.130
C09866=1110.595,-27.866,-50.326,179.768,5.938,149.131
C09867=1110.590,-27.617,-50.339,179.767,5.942,149.131
C09868=1110.585,-27.367,-50.352,179.767,5.947,149.133
C09869=1110.580,-27.117,-50.365,179.767,5.951,149.134
C09870=1110.575,-26.868,-50.377,179.767,5.955,149.135
C09871=1110.570,-26.618,-50.392,179.767,5.960,149.136
C09872=1110.565,-26.369,-50.404,179.767,5.964,149.136
C09873=1110.560,-26.120,-50.417,179.767,5.969,149.138
C09874=1110.555,-25.870,-50.430,179.767,5.973,149.138
C09875=1110.549,-25.620,-50.443,179.767,5.978,149.140
C09876=1110.544,-25.371,-50.456,179.767,5.983,149.141
C09877=1110.540,-25.121,-50.469,179.768,5.988,149.141
C09878=1110.534,-24.871,-50.482,179.768,5.992,149.142
C09879=1110.529,-24.622,-50.494,179.768,5.996,149.143
C09880=1110.523,-24.372,-50.508,179.769,6.001,149.144
C09881=1110.519,-24.123,-50.521,179.769,6.006,149.145
C09882=1110.514,-23.873,-50.534,179.769,6.011,149.146
C09883=1110.508,-23.623,-50.547,179.770,6.016,149.147
C09884=1110.503,-23.374,-50.560,179.770,6.020,149.148
C09885=1110.499,-23.124,-50.573,179.770,6.025,149.149
C09886=1110.493,-22.875,-50.587,179.771,6.030,149.150
C09887=1110.488,-22.625,-50.600,179.771,6.035,149.151
C09888=1110.483,-22.375,-50.613,179.772,6.039,149.152
C09889=1110.477,-22.126,-50.626,179.772,6.044,149.152
C09890=1110.472,-21.876,-50.639,179.773,6.049,149.153
C09891=1110.467,-21.627,-50.653,179.773,6.054,149.154
C09892=1110.463,-21.377,-50.666,179.774,6.058,149.155
C09893=1110.457,-21.127,-50.679,179.774,6.063,149.156
C09894=1110.452,-20.878,-50.691,179.775,6.068,149.157
C09895=1110.447,-20.628,-50.706,179.775,6.072,149.158
C09896=1110.442,-20.379,-50.718,179.776,6.077,149.159
C09897=1110.437,-20.129,-50.732,179.776,6.082,149.160
C09898=1110.432,-19.880,-50.745,179.777,6.087,149.161
C09899=1110.426,-19.630,-50.759,179.777,6.091,149.161
C09900=1110.421,-19.380,-50.771,179.777,6.095,149.162
C09901=1110.416,-19.130,-50.786,179.778,6.100,149.163
C09902=1110.411,-18.881,-50.798,179.779,6.104,149.164
C09903=1110.406,-18.667,-50.809,179.779,6.109,149.165
C09904=1110.403,-18.452,-50.822,179.779,6.113,149.166
C09905=1110.398,-18.237,-50.833,179.779,6.117,149.166
C09906=1110.394,-18.023,-50.844,179.780,6.121,149.167
C09907=1110.389,-17.809,-50.855,179.781,6.124,149.168
C09908=1110.385,-17.595,-50.867,179.781,6.128,149.169
C09909=1110.380,-17.379,-50.879,179.782,6.133,149.169
C09910=1110.376,-17.165,-50.890,179.782,6.136,149.170
C09911=1110.371,-16.916,-50.904,179.782,6.141,149.171
C09912=1110.366,-16.666,-50.917,179.783,6.146,149.172
C09913=1110.361,-16.417,-50.930,179.783,6.150,149.173
C09914=1110.355,-16.167,-50.944,179.784,6.155,149.174
C09915=1110.351,-15.918,-50.957,179.784,6.160,149.174
C09916=1110.345,-15.668,-50.971,179.785,6.164,149.175
C09917=1110.340,-15.419,-50.985,179.785,6.168,149.176
C09918=1110.335,-15.169,-50.998,179.786,6.173,149.177
C09919=1110.330,-14.919,-51.012,179.786,6.178,149.178
C09920=1110.325,-14.670,-51.025,179.787,6.182,149.179
C09921=1110.320,-14.420,-51.039,179.787,6.187,149.180
C09922=1110.314,-14.170,-51.052,179.788,6.191,149.180
C09923=1110.310,-13.921,-51.066,179.789,6.196,149.181
C09924=1110.304,-13.671,-51.079,179.789,6.201,149.182
C09925=1110.299,-13.422,-51.093,179.790,6.206,149.183
C09926=1110.295,-13.172,-51.106,179.790,6.210,149.184
C09927=1110.289,-12.923,-51.120,179.791,6.214,149.185
C09928=1110.284,-12.672,-51.134,179.791,6.219,149.185
C09929=1110.279,-12.424,-51.147,179.792,6.223,149.186
C09930=1110.274,-12.174,-51.161,179.792,6.228,149.187
C09931=1110.268,-11.924,-51.174,179.793,6.233,149.188
C09932=1110.264,-11.675,-51.188,179.794,6.237,149.189
C09933=1110.259,-11.425,-51.202,179.794,6.242,149.190
C09934=1110.253,-11.176,-51.216,179.795,6.247,149.191
C09935=1110.249,-10.926,-51.229,179.795,6.251,149.192
C09936=1110.244,-10.676,-51.243,179.795,6.255,149.192
C09937=1110.238,-10.427,-51.257,179.796,6.259,149.193
C09938=1110.234,-10.177,-51.270,179.796,6.264,149.194
C09939=1110.228,-9.928,-51.284,179.797,6.269,149.195
C09940=1110.223,-9.678,-51.298,179.798,6.273,149.196
C09941=1110.218,-9.428,-51.312,179.798,6.278,149.196
C09942=1110.214,-9.180,-51.325,179.799,6.283,149.197
C09943=1110.208,-8.929,-51.339,179.799,6.287,149.198
C09944=1110.203,-8.680,-51.353,179.800,6.292,149.199
C09945=1110.198,-8.431,-51.367,179.800,6.296,149.200
C09946=1110.193,-8.180,-51.381,179.801,6.300,149.201
C09947=1110.188,-7.931,-51.394,179.801,6.305,149.202
C09948=1110.183,-7.682,-51.408,179.802,6.309,149.202
C09949=1110.178,-7.432,-51.423,179.803,6.314,149.203
C09950=1110.173,-7.182,-51.437,179.803,6.319,149.204
C09951=1110.167,-6.933,-51.450,179.804,6.323,149.205
C09952=1110.163,-6.683,-51.464,179.805,6.328,149.206
C09953=1110.158,-6.434,-51.478,179.805,6.333,149.206
C09954=1110.152,-6.185,-51.492,179.805,6.337,149.207
C09955=1110.147,-5.935,-51.506,179.806,6.341,149.208
C09956=1110.142,-5.685,-51.520,179.807,6.346,149.209
C09957=1110.137,-5.435,-51.534,179.807,6.350,149.210
C09958=1110.132,-5.186,-51.547,179.808,6.355,149.210
C09959=1110.128,-4.971,-51.560,179.808,6.359,149.211
C09960=1110.123,-4.757,-51.572,179.809,6.363,149.212
C09961=1110.118,-4.543,-51.584,179.810,6.366,149.213
C09962=1110.115,-4.328,-51.596,179.810,6.370,149.213
C09963=1110.110,-4.114,-51.608,179.811,6.374,149.214
C09964=1110.106,-3.900,-51.621,179.811,6.378,149.215
C09965=1110.102,-3.686,-51.633,179.811,6.382,149.216
C09966=1110.097,-3.471,-51.644,179.812,6.386,149.216
C09967=1110.092,-3.221,-51.658,179.813,6.391,149.217
C09968=1110.087,-2.972,-51.673,179.813,6.394,149.218
C09969=1110.082,-2.722,-51.687,179.814,6.399,149.219
C09970=1110.077,-2.473,-51.701,179.814,6.404,149.220
C09971=1110.072,-2.223,-51.715,179.815,6.408,149.220
C09972=1110.067,-1.974,-51.729,179.816,6.413,149.221
C09973=1110.062,-1.724,-51.744,179.816,6.418,149.222
C09974=1110.056,-1.475,-51.757,179.817,6.422,149.223
C09975=1110.051,-1.225,-51.772,179.818,6.427,149.224
C09976=1110.046,-0.975,-51.786,179.818,6.431,149.225
C09977=1110.041,-0.726,-51.800,179.819,6.436,149.225
C09978=1110.036,-0.476,-51.815,179.820,6.440,149.226
C09979=1110.031,-0.227,-51.828,179.820,6.444,149.227
C09980=1110.026,0.023,-51.843,179.820,6.449,149.228
C09981=1110.021,0.272,-51.857,179.821,6.454,149.229
C09982=1110.016,0.521,-51.872,179.822,6.458,149.229
C09983=1110.011,0.771,-51.886,179.822,6.463,149.230
C09984=1110.006,1.021,-51.901,179.823,6.468,149.231
C09985=1110.001,1.270,-51.914,179.823,6.472,149.232
C09986=1109.996,1.520,-51.929,179.824,6.477,149.233
C09987=1109.991,1.769,-51.943,179.825,6.481,149.234
C09988=1109.986,2.019,-51.957,179.825,6.486,149.235
C09989=1109.981,2.269,-51.972,179.827,6.490,149.235
C09990=1109.976,2.518,-51.986,179.827,6.495,149.236
C09991=1109.971,2.767,-52.000,179.827,6.499,149.237
C09992=1109.966,3.017,-52.015,179.827,6.504,149.238
C09993=1109.961,3.266,-52.029,179.829,6.508,149.239
C09994=1109.956,3.516,-52.043,179.829,6.513,149.239
C09995=1109.951,3.766,-52.058,179.830,6.517,149.240
C09996=1109.946,4.015,-52.073,179.830,6.522,149.241
//INST
///DATE 2021/06/25 14:33
///ATTR SC,RW,RJ
////FRAME ROBOT
///GROUP1 RB1
NOP
MOVL C00000 V=800.0 PL=0
MOVL C00001 V=800.0 PL=0
MOVL C00002 V=800.0 PL=0
MOVL C00003 V=800.0 PL=0
MOVL C00004 V=800.0 PL=0
MOVL C00005 V=800.0 PL=0
MOVL C00006 V=800.0 PL=0
MOVL C00007 V=800.0 PL=0
MOVL C00008 V=800.0 PL=0
MOVL C00009 V=800.0 PL=0
MOVL C00010 V=800.0 PL=0
MOVL C00011 V=800.0 PL=0
MOVL C00012 V=800.0 PL=0
MOVL C00013 V=800.0 PL=0
MOVL C00014 V=800.0 PL=0
MOVL C00015 V=800.0 PL=0
MOVL C00016 V=800.0 PL=0
MOVL C00017 V=800.0 PL=0
MOVL C00018 V=800.0 PL=0
MOVL C00019 V=800.0 PL=0
MOVL C00020 V=800.0 PL=0
MOVL C00021 V=800.0 PL=0
MOVL C00022 V=800.0 PL=0
MOVL C00023 V=800.0 PL=0
MOVL C00024 V=800.0 PL=0
MOVL C00025 V=800.0 PL=0
MOVL C00026 V=800.0 PL=0
MOVL C00027 V=800.0 PL=0
MOVL C00028 V=800.0 PL=0
MOVL C00029 V=800.0 PL=0
MOVL C00030 V=800.0 PL=0
MOVL C00031 V=800.0 PL=0
MOVL C00032 V=800.0 PL=0
MOVL C00033 V=800.0 PL=0
MOVL C00034 V=800.0 PL=0
MOVL C00035 V=800.0 PL=0
MOVL C00036 V=800.0 PL=0
MOVL C00037 V=800.0 PL=0
MOVL C00038 V=800.0 PL=0
MOVL C00039 V=800.0 PL=0
MOVL C00040 V=800.0 PL=0
MOVL C00041 V=800.0 PL=0
MOVL C00042 V=800.0 PL=0
MOVL C00043 V=800.0 PL=0
MOVL C00044 V=800.0 PL=0
MOVL C00045 V=800.0 PL=0
MOVL C00046 V=800.0 PL=0
MOVL C00047 V=800.0 PL=0
MOVL C00048 V=800.0 PL=0
MOVL C00049 V=800.0 PL=0
MOVL C00050 V=800.0 PL=0
MOVL C00051 V=800.0 PL=0
MOVL C00052 V=800.0 PL=0
MOVL C00053 V=800.0 PL=0
MOVL C00054 V=800.0 PL=0
MOVL C00055 V=800.0 PL=0
MOVL C00056 V=800.0 PL=0
MOVL C00057 V=800.0 PL=0
MOVL C00058 V=800.0 PL=0
MOVL C00059 V=800.0 PL=0
MOVL C00060 V=800.0 PL=0
MOVL C00061 V=800.0 PL=0
MOVL C00062 V=800.0 PL=0
MOVL C00063 V=800.0 PL=0
MOVL C00064 V=800.0 PL=0
MOVL C00065 V=800.0 PL=0
MOVL C00066 V=800.0 PL=0
MOVL C00067 V=800.0 PL=0
MOVL C00068 V=800.0 PL=0
MOVL C00069 V=800.0 PL=0
MOVL C00070 V=800.0 PL=0
MOVL C00071 V=800.0 PL=0
MOVL C00072 V=800.0 PL=0
MOVL C00073 V=800.0 PL=0
MOVL C00074 V=800.0 PL=0
MOVL C00075 V=800.0 PL=0
MOVL C00076 V=800.0 PL=0
MOVL C00077 V=800.0 PL=0
MOVL C00078 V=800.0 PL=0
MOVL C00079 V=800.0 PL=0
MOVL C00080 V=800.0 PL=0
MOVL C00081 V=800.0 PL=0
MOVL C00082 V=800.0 PL=0
MOVL C00083 V=800.0 PL=0
MOVL C00084 V=800.0 PL=0
MOVL C00085 V=800.0 PL=0
MOVL C00086 V=800.0 PL=0
MOVL C00087 V=800.0 PL=0
MOVL C00088 V=800.0 PL=0
MOVL C00089 V=800.0 PL=0
MOVL C00090 V=800.0 PL=0
MOVL C00091 V=800.0 PL=0
MOVL C00092 V=800.0 PL=0
MOVL C00093 V=800.0 PL=0
MOVL C00094 V=800.0 PL=0
MOVL C00095 V=800.0 PL=0
MOVL C00096 V=800.0 PL=0
MOVL C00097 V=800.0 PL=0
MOVL C00098 V=800.0 PL=0
MOVL C00099 V=800.0 PL=0
MOVL C00100 V=800.0 PL=0
MOVL C00101 V=800.0 PL=0
MOVL C00102 V=800.0 PL=0
MOVL C00103 V=800.0 PL=0
MOVL C00104 V=800.0 PL=0
MOVL C00105 V=800.0 PL=0
MOVL C00106 V=800.0 PL=0
MOVL C00107 V=800.0 PL=0
MOVL C00108 V=800.0 PL=0
MOVL C00109 V=800.0 PL=0
MOVL C00110 V=800.0 PL=0
MOVL C00111 V=800.0 PL=0
MOVL C00112 V=800.0 PL=0
MOVL C00113 V=800.0 PL=0
MOVL C00114 V=800.0 PL=0
MOVL C00115 V=800.0 PL=0
MOVL C00116 V=800.0 PL=0
MOVL C00117 V=800.0 PL=0
MOVL C00118 V=800.0 PL=0
MOVL C00119 V=800.0 PL=0
MOVL C00120 V=800.0 PL=0
MOVL C00121 V=800.0 PL=0
MOVL C00122 V=800.0 PL=0
MOVL C00123 V=800.0 PL=0
MOVL C00124 V=800.0 PL=0
MOVL C00125 V=800.0 PL=0
MOVL C00126 V=800.0 PL=0
MOVL C00127 V=800.0 PL=0
MOVL C00128 V=800.0 PL=0
MOVL C00129 V=800.0 PL=0
MOVL C00130 V=800.0 PL=0
MOVL C00131 V=800.0 PL=0
MOVL C00132 V=800.0 PL=0
MOVL C00133 V=800.0 PL=0
MOVL C00134 V=800.0 PL=0
MOVL C00135 V=800.0 PL=0
MOVL C00136 V=800.0 PL=0
MOVL C00137 V=800.0 PL=0
MOVL C00138 V=800.0 PL=0
MOVL C00139 V=800.0 PL=0
MOVL C00140 V=800.0 PL=0
MOVL C00141 V=800.0 PL=0
MOVL C00142 V=800.0 PL=0
MOVL C00143 V=800.0 PL=0
MOVL C00144 V=800.0 PL=0
MOVL C00145 V=800.0 PL=0
MOVL C00146 V=800.0 PL=0
MOVL C00147 V=800.0 PL=0
MOVL C00148 V=800.0 PL=0
MOVL C00149 V=800.0 PL=0
MOVL C00150 V=800.0 PL=0
MOVL C00151 V=800.0 PL=0
MOVL C00152 V=800.0 PL=0
MOVL C00153 V=800.0 PL=0
MOVL C00154 V=800.0 PL=0
MOVL C00155 V=800.0 PL=0
MOVL C00156 V=800.0 PL=0
MOVL C00157 V=800.0 PL=0
MOVL C00158 V=800.0 PL=0
MOVL C00159 V=800.0 PL=0
MOVL C00160 V=800.0 PL=0
MOVL C00161 V=800.0 PL=0
MOVL C00162 V=800.0 PL=0
MOVL C00163 V=800.0 PL=0
MOVL C00164 V=800.0 PL=0
MOVL C00165 V=800.0 PL=0
MOVL C00166 V=800.0 PL=0
MOVL C00167 V=800.0 PL=0
MOVL C00168 V=800.0 PL=0
MOVL C00169 V=800.0 PL=0
MOVL C00170 V=800.0 PL=0
MOVL C00171 V=800.0 PL=0
MOVL C00172 V=800.0 PL=0
MOVL C00173 V=800.0 PL=0
MOVL C00174 V=800.0 PL=0
MOVL C00175 V=800.0 PL=0
MOVL C00176 V=800.0 PL=0
MOVL C00177 V=800.0 PL=0
MOVL C00178 V=800.0 PL=0
MOVL C00179 V=800.0 PL=0
MOVL C00180 V=800.0 PL=0
MOVL C00181 V=800.0 PL=0
MOVL C00182 V=800.0 PL=0
MOVL C00183 V=800.0 PL=0
MOVL C00184 V=800.0 PL=0
MOVL C00185 V=800.0 PL=0
MOVL C00186 V=800.0 PL=0
MOVL C00187 V=800.0 PL=0
MOVL C00188 V=800.0 PL=0
MOVL C00189 V=800.0 PL=0
MOVL C00190 V=800.0 PL=0
MOVL C00191 V=800.0 PL=0
MOVL C00192 V=800.0 PL=0
MOVL C00193 V=800.0 PL=0
MOVL C00194 V=800.0 PL=0
MOVL C00195 V=800.0 PL=0
MOVL C00196 V=800.0 PL=0
MOVL C00197 V=800.0 PL=0
MOVL C00198 V=800.0 PL=0
MOVL C00199 V=800.0 PL=0
MOVL C00200 V=800.0 PL=0
MOVL C00201 V=800.0 PL=0
MOVL C00202 V=800.0 PL=0
MOVL C00203 V=800.0 PL=0
MOVL C00204 V=800.0 PL=0
MOVL C00205 V=800.0 PL=0
MOVL C00206 V=800.0 PL=0
MOVL C00207 V=800.0 PL=0
MOVL C00208 V=800.0 PL=0
MOVL C00209 V=800.0 PL=0
MOVL C00210 V=800.0 PL=0
MOVL C00211 V=800.0 PL=0
MOVL C00212 V=800.0 PL=0
MOVL C00213 V=800.0 PL=0
MOVL C00214 V=800.0 PL=0
MOVL C00215 V=800.0 PL=0
MOVL C00216 V=800.0 PL=0
MOVL C00217 V=800.0 PL=0
MOVL C00218 V=800.0 PL=0
MOVL C00219 V=800.0 PL=0
MOVL C00220 V=800.0 PL=0
MOVL C00221 V=800.0 PL=0
MOVL C00222 V=800.0 PL=0
MOVL C00223 V=800.0 PL=0
MOVL C00224 V=800.0 PL=0
MOVL C00225 V=800.0 PL=0
MOVL C00226 V=800.0 PL=0
MOVL C00227 V=800.0 PL=0
MOVL C00228 V=800.0 PL=0
MOVL C00229 V=800.0 PL=0
MOVL C00230 V=800.0 PL=0
MOVL C00231 V=800.0 PL=0
MOVL C00232 V=800.0 PL=0
MOVL C00233 V=800.0 PL=0
MOVL C00234 V=800.0 PL=0
MOVL C00235 V=800.0 PL=0
MOVL C00236 V=800.0 PL=0
MOVL C00237 V=800.0 PL=0
MOVL C00238 V=800.0 PL=0
MOVL C00239 V=800.0 PL=0
MOVL C00240 V=800.0 PL=0
MOVL C00241 V=800.0 PL=0
MOVL C00242 V=800.0 PL=0
MOVL C00243 V=800.0 PL=0
MOVL C00244 V=800.0 PL=0
MOVL C00245 V=800.0 PL=0
MOVL C00246 V=800.0 PL=0
MOVL C00247 V=800.0 PL=0
MOVL C00248 V=800.0 PL=0
MOVL C00249 V=800.0 PL=0
MOVL C00250 V=800.0 PL=0
MOVL C00251 V=800.0 PL=0
MOVL C00252 V=800.0 PL=0
MOVL C00253 V=800.0 PL=0
MOVL C00254 V=800.0 PL=0
MOVL C00255 V=800.0 PL=0
MOVL C00256 V=800.0 PL=0
MOVL C00257 V=800.0 PL=0
MOVL C00258 V=800.0 PL=0
MOVL C00259 V=800.0 PL=0
MOVL C00260 V=800.0 PL=0
MOVL C00261 V=800.0 PL=0
MOVL C00262 V=800.0 PL=0
MOVL C00263 V=800.0 PL=0
MOVL C00264 V=800.0 PL=0
MOVL C00265 V=800.0 PL=0
MOVL C00266 V=800.0 PL=0
MOVL C00267 V=800.0 PL=0
MOVL C00268 V=800.0 PL=0
MOVL C00269 V=800.0 PL=0
MOVL C00270 V=800.0 PL=0
MOVL C00271 V=800.0 PL=0
MOVL C00272 V=800.0 PL=0
MOVL C00273 V=800.0 PL=0
MOVL C00274 V=800.0 PL=0
MOVL C00275 V=800.0 PL=0
MOVL C00276 V=800.0 PL=0
MOVL C00277 V=800.0 PL=0
MOVL C00278 V=800.0 PL=0
MOVL C00279 V=800.0 PL=0
MOVL C00280 V=800.0 PL=0
MOVL C00281 V=800.0 PL=0
MOVL C00282 V=800.0 PL=0
MOVL C00283 V=800.0 PL=0
MOVL C00284 V=800.0 PL=0
MOVL C00285 V=800.0 PL=0
MOVL C00286 V=800.0 PL=0
MOVL C00287 V=800.0 PL=0
MOVL C00288 V=800.0 PL=0
MOVL C00289 V=800.0 PL=0
MOVL C00290 V=800.0 PL=0
MOVL C00291 V=800.0 PL=0
MOVL C00292 V=800.0 PL=0
MOVL C00293 V=800.0 PL=0
MOVL C00294 V=800.0 PL=0
MOVL C00295 V=800.0 PL=0
MOVL C00296 V=800.0 PL=0
MOVL C00297 V=800.0 PL=0
MOVL C00298 V=800.0 PL=0
MOVL C00299 V=800.0 PL=0
MOVL C00300 V=800.0 PL=0
MOVL C00301 V=800.0 PL=0
MOVL C00302 V=800.0 PL=0
MOVL C00303 V=800.0 PL=0
MOVL C00304 V=800.0 PL=0
MOVL C00305 V=800.0 PL=0
MOVL C00306 V=800.0 PL=0
MOVL C00307 V=800.0 PL=0
MOVL C00308 V=800.0 PL=0
MOVL C00309 V=800.0 PL=0
MOVL C00310 V=800.0 PL=0
MOVL C00311 V=800.0 PL=0
MOVL C00312 V=800.0 PL=0
MOVL C00313 V=800.0 PL=0
MOVL C00314 V=800.0 PL=0
MOVL C00315 V=800.0 PL=0
MOVL C00316 V=800.0 PL=0
MOVL C00317 V=800.0 PL=0
MOVL C00318 V=800.0 PL=0
MOVL C00319 V=800.0 PL=0
MOVL C00320 V=800.0 PL=0
MOVL C00321 V=800.0 PL=0
MOVL C00322 V=800.0 PL=0
MOVL C00323 V=800.0 PL=0
MOVL C00324 V=800.0 PL=0
MOVL C00325 V=800.0 PL=0
MOVL C00326 V=800.0 PL=0
MOVL C00327 V=800.0 PL=0
MOVL C00328 V=800.0 PL=0
MOVL C00329 V=800.0 PL=0
MOVL C00330 V=800.0 PL=0
MOVL C00331 V=800.0 PL=0
MOVL C00332 V=800.0 PL=0
MOVL C00333 V=800.0 PL=0
MOVL C00334 V=800.0 PL=0
MOVL C00335 V=800.0 PL=0
MOVL C00336 V=800.0 PL=0
MOVL C00337 V=800.0 PL=0
MOVL C00338 V=800.0 PL=0
MOVL C00339 V=800.0 PL=0
MOVL C00340 V=800.0 PL=0
MOVL C00341 V=800.0 PL=0
MOVL C00342 V=800.0 PL=0
MOVL C00343 V=800.0 PL=0
MOVL C00344 V=800.0 PL=0
MOVL C00345 V=800.0 PL=0
MOVL C00346 V=800.0 PL=0
MOVL C00347 V=800.0 PL=0
MOVL C00348 V=800.0 PL=0
MOVL C00349 V=800.0 PL=0
MOVL C00350 V=800.0 PL=0
MOVL C00351 V=800.0 PL=0
MOVL C00352 V=800.0 PL=0
MOVL C00353 V=800.0 PL=0
MOVL C00354 V=800.0 PL=0
MOVL C00355 V=800.0 PL=0
MOVL C00356 V=800.0 PL=0
MOVL C00357 V=800.0 PL=0
MOVL C00358 V=800.0 PL=0
MOVL C00359 V=800.0 PL=0
MOVL C00360 V=800.0 PL=0
MOVL C00361 V=800.0 PL=0
MOVL C00362 V=800.0 PL=0
MOVL C00363 V=800.0 PL=0
MOVL C00364 V=800.0 PL=0
MOVL C00365 V=800.0 PL=0
MOVL C00366 V=800.0 PL=0
MOVL C00367 V=800.0 PL=0
MOVL C00368 V=800.0 PL=0
MOVL C00369 V=800.0 PL=0
MOVL C00370 V=800.0 PL=0
MOVL C00371 V=800.0 PL=0
MOVL C00372 V=800.0 PL=0
MOVL C00373 V=800.0 PL=0
MOVL C00374 V=800.0 PL=0
MOVL C00375 V=800.0 PL=0
MOVL C00376 V=800.0 PL=0
MOVL C00377 V=800.0 PL=0
MOVL C00378 V=800.0 PL=0
MOVL C00379 V=800.0 PL=0
MOVL C00380 V=800.0 PL=0
MOVL C00381 V=800.0 PL=0
MOVL C00382 V=800.0 PL=0
MOVL C00383 V=800.0 PL=0
MOVL C00384 V=800.0 PL=0
MOVL C00385 V=800.0 PL=0
MOVL C00386 V=800.0 PL=0
MOVL C00387 V=800.0 PL=0
MOVL C00388 V=800.0 PL=0
MOVL C00389 V=800.0 PL=0
MOVL C00390 V=800.0 PL=0
MOVL C00391 V=800.0 PL=0
MOVL C00392 V=800.0 PL=0
MOVL C00393 V=800.0 PL=0
MOVL C00394 V=800.0 PL=0
MOVL C00395 V=800.0 PL=0
MOVL C00396 V=800.0 PL=0
MOVL C00397 V=800.0 PL=0
MOVL C00398 V=800.0 PL=0
MOVL C00399 V=800.0 PL=0
MOVL C00400 V=800.0 PL=0
MOVL C00401 V=800.0 PL=0
MOVL C00402 V=800.0 PL=0
MOVL C00403 V=800.0 PL=0
MOVL C00404 V=800.0 PL=0
MOVL C00405 V=800.0 PL=0
MOVL C00406 V=800.0 PL=0
MOVL C00407 V=800.0 PL=0
MOVL C00408 V=800.0 PL=0
MOVL C00409 V=800.0 PL=0
MOVL C00410 V=800.0 PL=0
MOVL C00411 V=800.0 PL=0
MOVL C00412 V=800.0 PL=0
MOVL C00413 V=800.0 PL=0
MOVL C00414 V=800.0 PL=0
MOVL C00415 V=800.0 PL=0
MOVL C00416 V=800.0 PL=0
MOVL C00417 V=800.0 PL=0
MOVL C00418 V=800.0 PL=0
MOVL C00419 V=800.0 PL=0
MOVL C00420 V=800.0 PL=0
MOVL C00421 V=800.0 PL=0
MOVL C00422 V=800.0 PL=0
MOVL C00423 V=800.0 PL=0
MOVL C00424 V=800.0 PL=0
MOVL C00425 V=800.0 PL=0
MOVL C00426 V=800.0 PL=0
MOVL C00427 V=800.0 PL=0
MOVL C00428 V=800.0 PL=0
MOVL C00429 V=800.0 PL=0
MOVL C00430 V=800.0 PL=0
MOVL C00431 V=800.0 PL=0
MOVL C00432 V=800.0 PL=0
MOVL C00433 V=800.0 PL=0
MOVL C00434 V=800.0 PL=0
MOVL C00435 V=800.0 PL=0
MOVL C00436 V=800.0 PL=0
MOVL C00437 V=800.0 PL=0
MOVL C00438 V=800.0 PL=0
MOVL C00439 V=800.0 PL=0
MOVL C00440 V=800.0 PL=0
MOVL C00441 V=800.0 PL=0
MOVL C00442 V=800.0 PL=0
MOVL C00443 V=800.0 PL=0
MOVL C00444 V=800.0 PL=0
MOVL C00445 V=800.0 PL=0
MOVL C00446 V=800.0 PL=0
MOVL C00447 V=800.0 PL=0
MOVL C00448 V=800.0 PL=0
MOVL C00449 V=800.0 PL=0
MOVL C00450 V=800.0 PL=0
MOVL C00451 V=800.0 PL=0
MOVL C00452 V=800.0 PL=0
MOVL C00453 V=800.0 PL=0
MOVL C00454 V=800.0 PL=0
MOVL C00455 V=800.0 PL=0
MOVL C00456 V=800.0 PL=0
MOVL C00457 V=800.0 PL=0
MOVL C00458 V=800.0 PL=0
MOVL C00459 V=800.0 PL=0
MOVL C00460 V=800.0 PL=0
MOVL C00461 V=800.0 PL=0
MOVL C00462 V=800.0 PL=0
MOVL C00463 V=800.0 PL=0
MOVL C00464 V=800.0 PL=0
MOVL C00465 V=800.0 PL=0
MOVL C00466 V=800.0 PL=0
MOVL C00467 V=800.0 PL=0
MOVL C00468 V=800.0 PL=0
MOVL C00469 V=800.0 PL=0
MOVL C00470 V=800.0 PL=0
MOVL C00471 V=800.0 PL=0
MOVL C00472 V=800.0 PL=0
MOVL C00473 V=800.0 PL=0
MOVL C00474 V=800.0 PL=0
MOVL C00475 V=800.0 PL=0
MOVL C00476 V=800.0 PL=0
MOVL C00477 V=800.0 PL=0
MOVL C00478 V=800.0 PL=0
MOVL C00479 V=800.0 PL=0
MOVL C00480 V=800.0 PL=0
MOVL C00481 V=800.0 PL=0
MOVL C00482 V=800.0 PL=0
MOVL C00483 V=800.0 PL=0
MOVL C00484 V=800.0 PL=0
MOVL C00485 V=800.0 PL=0
MOVL C00486 V=800.0 PL=0
MOVL C00487 V=800.0 PL=0
MOVL C00488 V=800.0 PL=0
MOVL C00489 V=800.0 PL=0
MOVL C00490 V=800.0 PL=0
MOVL C00491 V=800.0 PL=0
MOVL C00492 V=800.0 PL=0
MOVL C00493 V=800.0 PL=0
MOVL C00494 V=800.0 PL=0
MOVL C00495 V=800.0 PL=0
MOVL C00496 V=800.0 PL=0
MOVL C00497 V=800.0 PL=0
MOVL C00498 V=800.0 PL=0
MOVL C00499 V=800.0 PL=0
MOVL C00500 V=800.0 PL=0
MOVL C00501 V=800.0 PL=0
MOVL C00502 V=800.0 PL=0
MOVL C00503 V=800.0 PL=0
MOVL C00504 V=800.0 PL=0
MOVL C00505 V=800.0 PL=0
MOVL C00506 V=800.0 PL=0
MOVL C00507 V=800.0 PL=0
MOVL C00508 V=800.0 PL=0
MOVL C00509 V=800.0 PL=0
MOVL C00510 V=800.0 PL=0
MOVL C00511 V=800.0 PL=0
MOVL C00512 V=800.0 PL=0
MOVL C00513 V=800.0 PL=0
MOVL C00514 V=800.0 PL=0
MOVL C00515 V=800.0 PL=0
MOVL C00516 V=800.0 PL=0
MOVL C00517 V=800.0 PL=0
MOVL C00518 V=800.0 PL=0
MOVL C00519 V=800.0 PL=0
MOVL C00520 V=800.0 PL=0
MOVL C00521 V=800.0 PL=0
MOVL C00522 V=800.0 PL=0
MOVL C00523 V=800.0 PL=0
MOVL C00524 V=800.0 PL=0
MOVL C00525 V=800.0 PL=0
MOVL C00526 V=800.0 PL=0
MOVL C00527 V=800.0 PL=0
MOVL C00528 V=800.0 PL=0
MOVL C00529 V=800.0 PL=0
MOVL C00530 V=800.0 PL=0
MOVL C00531 V=800.0 PL=0
MOVL C00532 V=800.0 PL=0
MOVL C00533 V=800.0 PL=0
MOVL C00534 V=800.0 PL=0
MOVL C00535 V=800.0 PL=0
MOVL C00536 V=800.0 PL=0
MOVL C00537 V=800.0 PL=0
MOVL C00538 V=800.0 PL=0
MOVL C00539 V=800.0 PL=0
MOVL C00540 V=800.0 PL=0
MOVL C00541 V=800.0 PL=0
MOVL C00542 V=800.0 PL=0
MOVL C00543 V=800.0 PL=0
MOVL C00544 V=800.0 PL=0
MOVL C00545 V=800.0 PL=0
MOVL C00546 V=800.0 PL=0
MOVL C00547 V=800.0 PL=0
MOVL C00548 V=800.0 PL=0
MOVL C00549 V=800.0 PL=0
MOVL C00550 V=800.0 PL=0
MOVL C00551 V=800.0 PL=0
MOVL C00552 V=800.0 PL=0
MOVL C00553 V=800.0 PL=0
MOVL C00554 V=800.0 PL=0
MOVL C00555 V=800.0 PL=0
MOVL C00556 V=800.0 PL=0
MOVL C00557 V=800.0 PL=0
MOVL C00558 V=800.0 PL=0
MOVL C00559 V=800.0 PL=0
MOVL C00560 V=800.0 PL=0
MOVL C00561 V=800.0 PL=0
MOVL C00562 V=800.0 PL=0
MOVL C00563 V=800.0 PL=0
MOVL C00564 V=800.0 PL=0
MOVL C00565 V=800.0 PL=0
MOVL C00566 V=800.0 PL=0
MOVL C00567 V=800.0 PL=0
MOVL C00568 V=800.0 PL=0
MOVL C00569 V=800.0 PL=0
MOVL C00570 V=800.0 PL=0
MOVL C00571 V=800.0 PL=0
MOVL C00572 V=800.0 PL=0
MOVL C00573 V=800.0 PL=0
MOVL C00574 V=800.0 PL=0
MOVL C00575 V=800.0 PL=0
MOVL C00576 V=800.0 PL=0
MOVL C00577 V=800.0 PL=0
MOVL C00578 V=800.0 PL=0
MOVL C00579 V=800.0 PL=0
MOVL C00580 V=800.0 PL=0
MOVL C00581 V=800.0 PL=0
MOVL C00582 V=800.0 PL=0
MOVL C00583 V=800.0 PL=0
MOVL C00584 V=800.0 PL=0
MOVL C00585 V=800.0 PL=0
MOVL C00586 V=800.0 PL=0
MOVL C00587 V=800.0 PL=0
MOVL C00588 V=800.0 PL=0
MOVL C00589 V=800.0 PL=0
MOVL C00590 V=800.0 PL=0
MOVL C00591 V=800.0 PL=0
MOVL C00592 V=800.0 PL=0
MOVL C00593 V=800.0 PL=0
MOVL C00594 V=800.0 PL=0
MOVL C00595 V=800.0 PL=0
MOVL C00596 V=800.0 PL=0
MOVL C00597 V=800.0 PL=0
MOVL C00598 V=800.0 PL=0
MOVL C00599 V=800.0 PL=0
MOVL C00600 V=800.0 PL=0
MOVL C00601 V=800.0 PL=0
MOVL C00602 V=800.0 PL=0
MOVL C00603 V=800.0 PL=0
MOVL C00604 V=800.0 PL=0
MOVL C00605 V=800.0 PL=0
MOVL C00606 V=800.0 PL=0
MOVL C00607 V=800.0 PL=0
MOVL C00608 V=800.0 PL=0
MOVL C00609 V=800.0 PL=0
MOVL C00610 V=800.0 PL=0
MOVL C00611 V=800.0 PL=0
MOVL C00612 V=800.0 PL=0
MOVL C00613 V=800.0 PL=0
MOVL C00614 V=800.0 PL=0
MOVL C00615 V=800.0 PL=0
MOVL C00616 V=800.0 PL=0
MOVL C00617 V=800.0 PL=0
MOVL C00618 V=800.0 PL=0
MOVL C00619 V=800.0 PL=0
MOVL C00620 V=800.0 PL=0
MOVL C00621 V=800.0 PL=0
MOVL C00622 V=800.0 PL=0
MOVL C00623 V=800.0 PL=0
MOVL C00624 V=800.0 PL=0
MOVL C00625 V=800.0 PL=0
MOVL C00626 V=800.0 PL=0
MOVL C00627 V=800.0 PL=0
MOVL C00628 V=800.0 PL=0
MOVL C00629 V=800.0 PL=0
MOVL C00630 V=800.0 PL=0
MOVL C00631 V=800.0 PL=0
MOVL C00632 V=800.0 PL=0
MOVL C00633 V=800.0 PL=0
MOVL C00634 V=800.0 PL=0
MOVL C00635 V=800.0 PL=0
MOVL C00636 V=800.0 PL=0
MOVL C00637 V=800.0 PL=0
MOVL C00638 V=800.0 PL=0
MOVL C00639 V=800.0 PL=0
MOVL C00640 V=800.0 PL=0
MOVL C00641 V=800.0 PL=0
MOVL C00642 V=800.0 PL=0
MOVL C00643 V=800.0 PL=0
MOVL C00644 V=800.0 PL=0
MOVL C00645 V=800.0 PL=0
MOVL C00646 V=800.0 PL=0
MOVL C00647 V=800.0 PL=0
MOVL C00648 V=800.0 PL=0
MOVL C00649 V=800.0 PL=0
MOVL C00650 V=800.0 PL=0
MOVL C00651 V=800.0 PL=0
MOVL C00652 V=800.0 PL=0
MOVL C00653 V=800.0 PL=0
MOVL C00654 V=800.0 PL=0
MOVL C00655 V=800.0 PL=0
MOVL C00656 V=800.0 PL=0
MOVL C00657 V=800.0 PL=0
MOVL C00658 V=800.0 PL=0
MOVL C00659 V=800.0 PL=0
MOVL C00660 V=800.0 PL=0
MOVL C00661 V=800.0 PL=0
MOVL C00662 V=800.0 PL=0
MOVL C00663 V=800.0 PL=0
MOVL C00664 V=800.0 PL=0
MOVL C00665 V=800.0 PL=0
MOVL C00666 V=800.0 PL=0
MOVL C00667 V=800.0 PL=0
MOVL C00668 V=800.0 PL=0
MOVL C00669 V=800.0 PL=0
MOVL C00670 V=800.0 PL=0
MOVL C00671 V=800.0 PL=0
MOVL C00672 V=800.0 PL=0
MOVL C00673 V=800.0 PL=0
MOVL C00674 V=800.0 PL=0
MOVL C00675 V=800.0 PL=0
MOVL C00676 V=800.0 PL=0
MOVL C00677 V=800.0 PL=0
MOVL C00678 V=800.0 PL=0
MOVL C00679 V=800.0 PL=0
MOVL C00680 V=800.0 PL=0
MOVL C00681 V=800.0 PL=0
MOVL C00682 V=800.0 PL=0
MOVL C00683 V=800.0 PL=0
MOVL C00684 V=800.0 PL=0
MOVL C00685 V=800.0 PL=0
MOVL C00686 V=800.0 PL=0
MOVL C00687 V=800.0 PL=0
MOVL C00688 V=800.0 PL=0
MOVL C00689 V=800.0 PL=0
MOVL C00690 V=800.0 PL=0
MOVL C00691 V=800.0 PL=0
MOVL C00692 V=800.0 PL=0
MOVL C00693 V=800.0 PL=0
MOVL C00694 V=800.0 PL=0
MOVL C00695 V=800.0 PL=0
MOVL C00696 V=800.0 PL=0
MOVL C00697 V=800.0 PL=0
MOVL C00698 V=800.0 PL=0
MOVL C00699 V=800.0 PL=0
MOVL C00700 V=800.0 PL=0
MOVL C00701 V=800.0 PL=0
MOVL C00702 V=800.0 PL=0
MOVL C00703 V=800.0 PL=0
MOVL C00704 V=800.0 PL=0
MOVL C00705 V=800.0 PL=0
MOVL C00706 V=800.0 PL=0
MOVL C00707 V=800.0 PL=0
MOVL C00708 V=800.0 PL=0
MOVL C00709 V=800.0 PL=0
MOVL C00710 V=800.0 PL=0
MOVL C00711 V=800.0 PL=0
MOVL C00712 V=800.0 PL=0
MOVL C00713 V=800.0 PL=0
MOVL C00714 V=800.0 PL=0
MOVL C00715 V=800.0 PL=0
MOVL C00716 V=800.0 PL=0
MOVL C00717 V=800.0 PL=0
MOVL C00718 V=800.0 PL=0
MOVL C00719 V=800.0 PL=0
MOVL C00720 V=800.0 PL=0
MOVL C00721 V=800.0 PL=0
MOVL C00722 V=800.0 PL=0
MOVL C00723 V=800.0 PL=0
MOVL C00724 V=800.0 PL=0
MOVL C00725 V=800.0 PL=0
MOVL C00726 V=800.0 PL=0
MOVL C00727 V=800.0 PL=0
MOVL C00728 V=800.0 PL=0
MOVL C00729 V=800.0 PL=0
MOVL C00730 V=800.0 PL=0
MOVL C00731 V=800.0 PL=0
MOVL C00732 V=800.0 PL=0
MOVL C00733 V=800.0 PL=0
MOVL C00734 V=800.0 PL=0
MOVL C00735 V=800.0 PL=0
MOVL C00736 V=800.0 PL=0
MOVL C00737 V=800.0 PL=0
MOVL C00738 V=800.0 PL=0
MOVL C00739 V=800.0 PL=0
MOVL C00740 V=800.0 PL=0
MOVL C00741 V=800.0 PL=0
MOVL C00742 V=800.0 PL=0
MOVL C00743 V=800.0 PL=0
MOVL C00744 V=800.0 PL=0
MOVL C00745 V=800.0 PL=0
MOVL C00746 V=800.0 PL=0
MOVL C00747 V=800.0 PL=0
MOVL C00748 V=800.0 PL=0
MOVL C00749 V=800.0 PL=0
MOVL C00750 V=800.0 PL=0
MOVL C00751 V=800.0 PL=0
MOVL C00752 V=800.0 PL=0
MOVL C00753 V=800.0 PL=0
MOVL C00754 V=800.0 PL=0
MOVL C00755 V=800.0 PL=0
MOVL C00756 V=800.0 PL=0
MOVL C00757 V=800.0 PL=0
MOVL C00758 V=800.0 PL=0
MOVL C00759 V=800.0 PL=0
MOVL C00760 V=800.0 PL=0
MOVL C00761 V=800.0 PL=0
MOVL C00762 V=800.0 PL=0
MOVL C00763 V=800.0 PL=0
MOVL C00764 V=800.0 PL=0
MOVL C00765 V=800.0 PL=0
MOVL C00766 V=800.0 PL=0
MOVL C00767 V=800.0 PL=0
MOVL C00768 V=800.0 PL=0
MOVL C00769 V=800.0 PL=0
MOVL C00770 V=800.0 PL=0
MOVL C00771 V=800.0 PL=0
MOVL C00772 V=800.0 PL=0
MOVL C00773 V=800.0 PL=0
MOVL C00774 V=800.0 PL=0
MOVL C00775 V=800.0 PL=0
MOVL C00776 V=800.0 PL=0
MOVL C00777 V=800.0 PL=0
MOVL C00778 V=800.0 PL=0
MOVL C00779 V=800.0 PL=0
MOVL C00780 V=800.0 PL=0
MOVL C00781 V=800.0 PL=0
MOVL C00782 V=800.0 PL=0
MOVL C00783 V=800.0 PL=0
MOVL C00784 V=800.0 PL=0
MOVL C00785 V=800.0 PL=0
MOVL C00786 V=800.0 PL=0
MOVL C00787 V=800.0 PL=0
MOVL C00788 V=800.0 PL=0
MOVL C00789 V=800.0 PL=0
MOVL C00790 V=800.0 PL=0
MOVL C00791 V=800.0 PL=0
MOVL C00792 V=800.0 PL=0
MOVL C00793 V=800.0 PL=0
MOVL C00794 V=800.0 PL=0
MOVL C00795 V=800.0 PL=0
MOVL C00796 V=800.0 PL=0
MOVL C00797 V=800.0 PL=0
MOVL C00798 V=800.0 PL=0
MOVL C00799 V=800.0 PL=0
MOVL C00800 V=800.0 PL=0
MOVL C00801 V=800.0 PL=0
MOVL C00802 V=800.0 PL=0
MOVL C00803 V=800.0 PL=0
MOVL C00804 V=800.0 PL=0
MOVL C00805 V=800.0 PL=0
MOVL C00806 V=800.0 PL=0
MOVL C00807 V=800.0 PL=0
MOVL C00808 V=800.0 PL=0
MOVL C00809 V=800.0 PL=0
MOVL C00810 V=800.0 PL=0
MOVL C00811 V=800.0 PL=0
MOVL C00812 V=800.0 PL=0
MOVL C00813 V=800.0 PL=0
MOVL C00814 V=800.0 PL=0
MOVL C00815 V=800.0 PL=0
MOVL C00816 V=800.0 PL=0
MOVL C00817 V=800.0 PL=0
MOVL C00818 V=800.0 PL=0
MOVL C00819 V=800.0 PL=0
MOVL C00820 V=800.0 PL=0
MOVL C00821 V=800.0 PL=0
MOVL C00822 V=800.0 PL=0
MOVL C00823 V=800.0 PL=0
MOVL C00824 V=800.0 PL=0
MOVL C00825 V=800.0 PL=0
MOVL C00826 V=800.0 PL=0
MOVL C00827 V=800.0 PL=0
MOVL C00828 V=800.0 PL=0
MOVL C00829 V=800.0 PL=0
MOVL C00830 V=800.0 PL=0
MOVL C00831 V=800.0 PL=0
MOVL C00832 V=800.0 PL=0
MOVL C00833 V=800.0 PL=0
MOVL C00834 V=800.0 PL=0
MOVL C00835 V=800.0 PL=0
MOVL C00836 V=800.0 PL=0
MOVL C00837 V=800.0 PL=0
MOVL C00838 V=800.0 PL=0
MOVL C00839 V=800.0 PL=0
MOVL C00840 V=800.0 PL=0
MOVL C00841 V=800.0 PL=0
MOVL C00842 V=800.0 PL=0
MOVL C00843 V=800.0 PL=0
MOVL C00844 V=800.0 PL=0
MOVL C00845 V=800.0 PL=0
MOVL C00846 V=800.0 PL=0
MOVL C00847 V=800.0 PL=0
MOVL C00848 V=800.0 PL=0
MOVL C00849 V=800.0 PL=0
MOVL C00850 V=800.0 PL=0
MOVL C00851 V=800.0 PL=0
MOVL C00852 V=800.0 PL=0
MOVL C00853 V=800.0 PL=0
MOVL C00854 V=800.0 PL=0
MOVL C00855 V=800.0 PL=0
MOVL C00856 V=800.0 PL=0
MOVL C00857 V=800.0 PL=0
MOVL C00858 V=800.0 PL=0
MOVL C00859 V=800.0 PL=0
MOVL C00860 V=800.0 PL=0
MOVL C00861 V=800.0 PL=0
MOVL C00862 V=800.0 PL=0
MOVL C00863 V=800.0 PL=0
MOVL C00864 V=800.0 PL=0
MOVL C00865 V=800.0 PL=0
MOVL C00866 V=800.0 PL=0
MOVL C00867 V=800.0 PL=0
MOVL C00868 V=800.0 PL=0
MOVL C00869 V=800.0 PL=0
MOVL C00870 V=800.0 PL=0
MOVL C00871 V=800.0 PL=0
MOVL C00872 V=800.0 PL=0
MOVL C00873 V=800.0 PL=0
MOVL C00874 V=800.0 PL=0
MOVL C00875 V=800.0 PL=0
MOVL C00876 V=800.0 PL=0
MOVL C00877 V=800.0 PL=0
MOVL C00878 V=800.0 PL=0
MOVL C00879 V=800.0 PL=0
MOVL C00880 V=800.0 PL=0
MOVL C00881 V=800.0 PL=0
MOVL C00882 V=800.0 PL=0
MOVL C00883 V=800.0 PL=0
MOVL C00884 V=800.0 PL=0
MOVL C00885 V=800.0 PL=0
MOVL C00886 V=800.0 PL=0
MOVL C00887 V=800.0 PL=0
MOVL C00888 V=800.0 PL=0
MOVL C00889 V=800.0 PL=0
MOVL C00890 V=800.0 PL=0
MOVL C00891 V=800.0 PL=0
MOVL C00892 V=800.0 PL=0
MOVL C00893 V=800.0 PL=0
MOVL C00894 V=800.0 PL=0
MOVL C00895 V=800.0 PL=0
MOVL C00896 V=800.0 PL=0
MOVL C00897 V=800.0 PL=0
MOVL C00898 V=800.0 PL=0
MOVL C00899 V=800.0 PL=0
MOVL C00900 V=800.0 PL=0
MOVL C00901 V=800.0 PL=0
MOVL C00902 V=800.0 PL=0
MOVL C00903 V=800.0 PL=0
MOVL C00904 V=800.0 PL=0
MOVL C00905 V=800.0 PL=0
MOVL C00906 V=800.0 PL=0
MOVL C00907 V=800.0 PL=0
MOVL C00908 V=800.0 PL=0
MOVL C00909 V=800.0 PL=0
MOVL C00910 V=800.0 PL=0
MOVL C00911 V=800.0 PL=0
MOVL C00912 V=800.0 PL=0
MOVL C00913 V=800.0 PL=0
MOVL C00914 V=800.0 PL=0
MOVL C00915 V=800.0 PL=0
MOVL C00916 V=800.0 PL=0
MOVL C00917 V=800.0 PL=0
MOVL C00918 V=800.0 PL=0
MOVL C00919 V=800.0 PL=0
MOVL C00920 V=800.0 PL=0
MOVL C00921 V=800.0 PL=0
MOVL C00922 V=800.0 PL=0
MOVL C00923 V=800.0 PL=0
MOVL C00924 V=800.0 PL=0
MOVL C00925 V=800.0 PL=0
MOVL C00926 V=800.0 PL=0
MOVL C00927 V=800.0 PL=0
MOVL C00928 V=800.0 PL=0
MOVL C00929 V=800.0 PL=0
MOVL C00930 V=800.0 PL=0
MOVL C00931 V=800.0 PL=0
MOVL C00932 V=800.0 PL=0
MOVL C00933 V=800.0 PL=0
MOVL C00934 V=800.0 PL=0
MOVL C00935 V=800.0 PL=0
MOVL C00936 V=800.0 PL=0
MOVL C00937 V=800.0 PL=0
MOVL C00938 V=800.0 PL=0
MOVL C00939 V=800.0 PL=0
MOVL C00940 V=800.0 PL=0
MOVL C00941 V=800.0 PL=0
MOVL C00942 V=800.0 PL=0
MOVL C00943 V=800.0 PL=0
MOVL C00944 V=800.0 PL=0
MOVL C00945 V=800.0 PL=0
MOVL C00946 V=800.0 PL=0
MOVL C00947 V=800.0 PL=0
MOVL C00948 V=800.0 PL=0
MOVL C00949 V=800.0 PL=0
MOVL C00950 V=800.0 PL=0
MOVL C00951 V=800.0 PL=0
MOVL C00952 V=800.0 PL=0
MOVL C00953 V=800.0 PL=0
MOVL C00954 V=800.0 PL=0
MOVL C00955 V=800.0 PL=0
MOVL C00956 V=800.0 PL=0
MOVL C00957 V=800.0 PL=0
MOVL C00958 V=800.0 PL=0
MOVL C00959 V=800.0 PL=0
MOVL C00960 V=800.0 PL=0
MOVL C00961 V=800.0 PL=0
MOVL C00962 V=800.0 PL=0
MOVL C00963 V=800.0 PL=0
MOVL C00964 V=800.0 PL=0
MOVL C00965 V=800.0 PL=0
MOVL C00966 V=800.0 PL=0
MOVL C00967 V=800.0 PL=0
MOVL C00968 V=800.0 PL=0
MOVL C00969 V=800.0 PL=0
MOVL C00970 V=800.0 PL=0
MOVL C00971 V=800.0 PL=0
MOVL C00972 V=800.0 PL=0
MOVL C00973 V=800.0 PL=0
MOVL C00974 V=800.0 PL=0
MOVL C00975 V=800.0 PL=0
MOVL C00976 V=800.0 PL=0
MOVL C00977 V=800.0 PL=0
MOVL C00978 V=800.0 PL=0
MOVL C00979 V=800.0 PL=0
MOVL C00980 V=800.0 PL=0
MOVL C00981 V=800.0 PL=0
MOVL C00982 V=800.0 PL=0
MOVL C00983 V=800.0 PL=0
MOVL C00984 V=800.0 PL=0
MOVL C00985 V=800.0 PL=0
MOVL C00986 V=800.0 PL=0
MOVL C00987 V=800.0 PL=0
MOVL C00988 V=800.0 PL=0
MOVL C00989 V=800.0 PL=0
MOVL C00990 V=800.0 PL=0
MOVL C00991 V=800.0 PL=0
MOVL C00992 V=800.0 PL=0
MOVL C00993 V=800.0 PL=0
MOVL C00994 V=800.0 PL=0
MOVL C00995 V=800.0 PL=0
MOVL C00996 V=800.0 PL=0
MOVL C00997 V=800.0 PL=0
MOVL C00998 V=800.0 PL=0
MOVL C00999 V=800.0 PL=0
MOVL C01000 V=800.0 PL=0
MOVL C01001 V=800.0 PL=0
MOVL C01002 V=800.0 PL=0
MOVL C01003 V=800.0 PL=0
MOVL C01004 V=800.0 PL=0
MOVL C01005 V=800.0 PL=0
MOVL C01006 V=800.0 PL=0
MOVL C01007 V=800.0 PL=0
MOVL C01008 V=800.0 PL=0
MOVL C01009 V=800.0 PL=0
MOVL C01010 V=800.0 PL=0
MOVL C01011 V=800.0 PL=0
MOVL C01012 V=800.0 PL=0
MOVL C01013 V=800.0 PL=0
MOVL C01014 V=800.0 PL=0
MOVL C01015 V=800.0 PL=0
MOVL C01016 V=800.0 PL=0
MOVL C01017 V=800.0 PL=0
MOVL C01018 V=800.0 PL=0
MOVL C01019 V=800.0 PL=0
MOVL C01020 V=800.0 PL=0
MOVL C01021 V=800.0 PL=0
MOVL C01022 V=800.0 PL=0
MOVL C01023 V=800.0 PL=0
MOVL C01024 V=800.0 PL=0
MOVL C01025 V=800.0 PL=0
MOVL C01026 V=800.0 PL=0
MOVL C01027 V=800.0 PL=0
MOVL C01028 V=800.0 PL=0
MOVL C01029 V=800.0 PL=0
MOVL C01030 V=800.0 PL=0
MOVL C01031 V=800.0 PL=0
MOVL C01032 V=800.0 PL=0
MOVL C01033 V=800.0 PL=0
MOVL C01034 V=800.0 PL=0
MOVL C01035 V=800.0 PL=0
MOVL C01036 V=800.0 PL=0
MOVL C01037 V=800.0 PL=0
MOVL C01038 V=800.0 PL=0
MOVL C01039 V=800.0 PL=0
MOVL C01040 V=800.0 PL=0
MOVL C01041 V=800.0 PL=0
MOVL C01042 V=800.0 PL=0
MOVL C01043 V=800.0 PL=0
MOVL C01044 V=800.0 PL=0
MOVL C01045 V=800.0 PL=0
MOVL C01046 V=800.0 PL=0
MOVL C01047 V=800.0 PL=0
MOVL C01048 V=800.0 PL=0
MOVL C01049 V=800.0 PL=0
MOVL C01050 V=800.0 PL=0
MOVL C01051 V=800.0 PL=0
MOVL C01052 V=800.0 PL=0
MOVL C01053 V=800.0 PL=0
MOVL C01054 V=800.0 PL=0
MOVL C01055 V=800.0 PL=0
MOVL C01056 V=800.0 PL=0
MOVL C01057 V=800.0 PL=0
MOVL C01058 V=800.0 PL=0
MOVL C01059 V=800.0 PL=0
MOVL C01060 V=800.0 PL=0
MOVL C01061 V=800.0 PL=0
MOVL C01062 V=800.0 PL=0
MOVL C01063 V=800.0 PL=0
MOVL C01064 V=800.0 PL=0
MOVL C01065 V=800.0 PL=0
MOVL C01066 V=800.0 PL=0
MOVL C01067 V=800.0 PL=0
MOVL C01068 V=800.0 PL=0
MOVL C01069 V=800.0 PL=0
MOVL C01070 V=800.0 PL=0
MOVL C01071 V=800.0 PL=0
MOVL C01072 V=800.0 PL=0
MOVL C01073 V=800.0 PL=0
MOVL C01074 V=800.0 PL=0
MOVL C01075 V=800.0 PL=0
MOVL C01076 V=800.0 PL=0
MOVL C01077 V=800.0 PL=0
MOVL C01078 V=800.0 PL=0
MOVL C01079 V=800.0 PL=0
MOVL C01080 V=800.0 PL=0
MOVL C01081 V=800.0 PL=0
MOVL C01082 V=800.0 PL=0
MOVL C01083 V=800.0 PL=0
MOVL C01084 V=800.0 PL=0
MOVL C01085 V=800.0 PL=0
MOVL C01086 V=800.0 PL=0
MOVL C01087 V=800.0 PL=0
MOVL C01088 V=800.0 PL=0
MOVL C01089 V=800.0 PL=0
MOVL C01090 V=800.0 PL=0
MOVL C01091 V=800.0 PL=0
MOVL C01092 V=800.0 PL=0
MOVL C01093 V=800.0 PL=0
MOVL C01094 V=800.0 PL=0
MOVL C01095 V=800.0 PL=0
MOVL C01096 V=800.0 PL=0
MOVL C01097 V=800.0 PL=0
MOVL C01098 V=800.0 PL=0
MOVL C01099 V=800.0 PL=0
MOVL C01100 V=800.0 PL=0
MOVL C01101 V=800.0 PL=0
MOVL C01102 V=800.0 PL=0
MOVL C01103 V=800.0 PL=0
MOVL C01104 V=800.0 PL=0
MOVL C01105 V=800.0 PL=0
MOVL C01106 V=800.0 PL=0
MOVL C01107 V=800.0 PL=0
MOVL C01108 V=800.0 PL=0
MOVL C01109 V=800.0 PL=0
MOVL C01110 V=800.0 PL=0
MOVL C01111 V=800.0 PL=0
MOVL C01112 V=800.0 PL=0
MOVL C01113 V=800.0 PL=0
MOVL C01114 V=800.0 PL=0
MOVL C01115 V=800.0 PL=0
MOVL C01116 V=800.0 PL=0
MOVL C01117 V=800.0 PL=0
MOVL C01118 V=800.0 PL=0
MOVL C01119 V=800.0 PL=0
MOVL C01120 V=800.0 PL=0
MOVL C01121 V=800.0 PL=0
MOVL C01122 V=800.0 PL=0
MOVL C01123 V=800.0 PL=0
MOVL C01124 V=800.0 PL=0
MOVL C01125 V=800.0 PL=0
MOVL C01126 V=800.0 PL=0
MOVL C01127 V=800.0 PL=0
MOVL C01128 V=800.0 PL=0
MOVL C01129 V=800.0 PL=0
MOVL C01130 V=800.0 PL=0
MOVL C01131 V=800.0 PL=0
MOVL C01132 V=800.0 PL=0
MOVL C01133 V=800.0 PL=0
MOVL C01134 V=800.0 PL=0
MOVL C01135 V=800.0 PL=0
MOVL C01136 V=800.0 PL=0
MOVL C01137 V=800.0 PL=0
MOVL C01138 V=800.0 PL=0
MOVL C01139 V=800.0 PL=0
MOVL C01140 V=800.0 PL=0
MOVL C01141 V=800.0 PL=0
MOVL C01142 V=800.0 PL=0
MOVL C01143 V=800.0 PL=0
MOVL C01144 V=800.0 PL=0
MOVL C01145 V=800.0 PL=0
MOVL C01146 V=800.0 PL=0
MOVL C01147 V=800.0 PL=0
MOVL C01148 V=800.0 PL=0
MOVL C01149 V=800.0 PL=0
MOVL C01150 V=800.0 PL=0
MOVL C01151 V=800.0 PL=0
MOVL C01152 V=800.0 PL=0
MOVL C01153 V=800.0 PL=0
MOVL C01154 V=800.0 PL=0
MOVL C01155 V=800.0 PL=0
MOVL C01156 V=800.0 PL=0
MOVL C01157 V=800.0 PL=0
MOVL C01158 V=800.0 PL=0
MOVL C01159 V=800.0 PL=0
MOVL C01160 V=800.0 PL=0
MOVL C01161 V=800.0 PL=0
MOVL C01162 V=800.0 PL=0
MOVL C01163 V=800.0 PL=0
MOVL C01164 V=800.0 PL=0
MOVL C01165 V=800.0 PL=0
MOVL C01166 V=800.0 PL=0
MOVL C01167 V=800.0 PL=0
MOVL C01168 V=800.0 PL=0
MOVL C01169 V=800.0 PL=0
MOVL C01170 V=800.0 PL=0
MOVL C01171 V=800.0 PL=0
MOVL C01172 V=800.0 PL=0
MOVL C01173 V=800.0 PL=0
MOVL C01174 V=800.0 PL=0
MOVL C01175 V=800.0 PL=0
MOVL C01176 V=800.0 PL=0
MOVL C01177 V=800.0 PL=0
MOVL C01178 V=800.0 PL=0
MOVL C01179 V=800.0 PL=0
MOVL C01180 V=800.0 PL=0
MOVL C01181 V=800.0 PL=0
MOVL C01182 V=800.0 PL=0
MOVL C01183 V=800.0 PL=0
MOVL C01184 V=800.0 PL=0
MOVL C01185 V=800.0 PL=0
MOVL C01186 V=800.0 PL=0
MOVL C01187 V=800.0 PL=0
MOVL C01188 V=800.0 PL=0
MOVL C01189 V=800.0 PL=0
MOVL C01190 V=800.0 PL=0
MOVL C01191 V=800.0 PL=0
MOVL C01192 V=800.0 PL=0
MOVL C01193 V=800.0 PL=0
MOVL C01194 V=800.0 PL=0
MOVL C01195 V=800.0 PL=0
MOVL C01196 V=800.0 PL=0
MOVL C01197 V=800.0 PL=0
MOVL C01198 V=800.0 PL=0
MOVL C01199 V=800.0 PL=0
MOVL C01200 V=800.0 PL=0
MOVL C01201 V=800.0 PL=0
MOVL C01202 V=800.0 PL=0
MOVL C01203 V=800.0 PL=0
MOVL C01204 V=800.0 PL=0
MOVL C01205 V=800.0 PL=0
MOVL C01206 V=800.0 PL=0
MOVL C01207 V=800.0 PL=0
MOVL C01208 V=800.0 PL=0
MOVL C01209 V=800.0 PL=0
MOVL C01210 V=800.0 PL=0
MOVL C01211 V=800.0 PL=0
MOVL C01212 V=800.0 PL=0
MOVL C01213 V=800.0 PL=0
MOVL C01214 V=800.0 PL=0
MOVL C01215 V=800.0 PL=0
MOVL C01216 V=800.0 PL=0
MOVL C01217 V=800.0 PL=0
MOVL C01218 V=800.0 PL=0
MOVL C01219 V=800.0 PL=0
MOVL C01220 V=800.0 PL=0
MOVL C01221 V=800.0 PL=0
MOVL C01222 V=800.0 PL=0
MOVL C01223 V=800.0 PL=0
MOVL C01224 V=800.0 PL=0
MOVL C01225 V=800.0 PL=0
MOVL C01226 V=800.0 PL=0
MOVL C01227 V=800.0 PL=0
MOVL C01228 V=800.0 PL=0
MOVL C01229 V=800.0 PL=0
MOVL C01230 V=800.0 PL=0
MOVL C01231 V=800.0 PL=0
MOVL C01232 V=800.0 PL=0
MOVL C01233 V=800.0 PL=0
MOVL C01234 V=800.0 PL=0
MOVL C01235 V=800.0 PL=0
MOVL C01236 V=800.0 PL=0
MOVL C01237 V=800.0 PL=0
MOVL C01238 V=800.0 PL=0
MOVL C01239 V=800.0 PL=0
MOVL C01240 V=800.0 PL=0
MOVL C01241 V=800.0 PL=0
MOVL C01242 V=800.0 PL=0
MOVL C01243 V=800.0 PL=0
MOVL C01244 V=800.0 PL=0
MOVL C01245 V=800.0 PL=0
MOVL C01246 V=800.0 PL=0
MOVL C01247 V=800.0 PL=0
MOVL C01248 V=800.0 PL=0
MOVL C01249 V=800.0 PL=0
MOVL C01250 V=800.0 PL=0
MOVL C01251 V=800.0 PL=0
MOVL C01252 V=800.0 PL=0
MOVL C01253 V=800.0 PL=0
MOVL C01254 V=800.0 PL=0
MOVL C01255 V=800.0 PL=0
MOVL C01256 V=800.0 PL=0
MOVL C01257 V=800.0 PL=0
MOVL C01258 V=800.0 PL=0
MOVL C01259 V=800.0 PL=0
MOVL C01260 V=800.0 PL=0
MOVL C01261 V=800.0 PL=0
MOVL C01262 V=800.0 PL=0
MOVL C01263 V=800.0 PL=0
MOVL C01264 V=800.0 PL=0
MOVL C01265 V=800.0 PL=0
MOVL C01266 V=800.0 PL=0
MOVL C01267 V=800.0 PL=0
MOVL C01268 V=800.0 PL=0
MOVL C01269 V=800.0 PL=0
MOVL C01270 V=800.0 PL=0
MOVL C01271 V=800.0 PL=0
MOVL C01272 V=800.0 PL=0
MOVL C01273 V=800.0 PL=0
MOVL C01274 V=800.0 PL=0
MOVL C01275 V=800.0 PL=0
MOVL C01276 V=800.0 PL=0
MOVL C01277 V=800.0 PL=0
MOVL C01278 V=800.0 PL=0
MOVL C01279 V=800.0 PL=0
MOVL C01280 V=800.0 PL=0
MOVL C01281 V=800.0 PL=0
MOVL C01282 V=800.0 PL=0
MOVL C01283 V=800.0 PL=0
MOVL C01284 V=800.0 PL=0
MOVL C01285 V=800.0 PL=0
MOVL C01286 V=800.0 PL=0
MOVL C01287 V=800.0 PL=0
MOVL C01288 V=800.0 PL=0
MOVL C01289 V=800.0 PL=0
MOVL C01290 V=800.0 PL=0
MOVL C01291 V=800.0 PL=0
MOVL C01292 V=800.0 PL=0
MOVL C01293 V=800.0 PL=0
MOVL C01294 V=800.0 PL=0
MOVL C01295 V=800.0 PL=0
MOVL C01296 V=800.0 PL=0
MOVL C01297 V=800.0 PL=0
MOVL C01298 V=800.0 PL=0
MOVL C01299 V=800.0 PL=0
MOVL C01300 V=800.0 PL=0
MOVL C01301 V=800.0 PL=0
MOVL C01302 V=800.0 PL=0
MOVL C01303 V=800.0 PL=0
MOVL C01304 V=800.0 PL=0
MOVL C01305 V=800.0 PL=0
MOVL C01306 V=800.0 PL=0
MOVL C01307 V=800.0 PL=0
MOVL C01308 V=800.0 PL=0
MOVL C01309 V=800.0 PL=0
MOVL C01310 V=800.0 PL=0
MOVL C01311 V=800.0 PL=0
MOVL C01312 V=800.0 PL=0
MOVL C01313 V=800.0 PL=0
MOVL C01314 V=800.0 PL=0
MOVL C01315 V=800.0 PL=0
MOVL C01316 V=800.0 PL=0
MOVL C01317 V=800.0 PL=0
MOVL C01318 V=800.0 PL=0
MOVL C01319 V=800.0 PL=0
MOVL C01320 V=800.0 PL=0
MOVL C01321 V=800.0 PL=0
MOVL C01322 V=800.0 PL=0
MOVL C01323 V=800.0 PL=0
MOVL C01324 V=800.0 PL=0
MOVL C01325 V=800.0 PL=0
MOVL C01326 V=800.0 PL=0
MOVL C01327 V=800.0 PL=0
MOVL C01328 V=800.0 PL=0
MOVL C01329 V=800.0 PL=0
MOVL C01330 V=800.0 PL=0
MOVL C01331 V=800.0 PL=0
MOVL C01332 V=800.0 PL=0
MOVL C01333 V=800.0 PL=0
MOVL C01334 V=800.0 PL=0
MOVL C01335 V=800.0 PL=0
MOVL C01336 V=800.0 PL=0
MOVL C01337 V=800.0 PL=0
MOVL C01338 V=800.0 PL=0
MOVL C01339 V=800.0 PL=0
MOVL C01340 V=800.0 PL=0
MOVL C01341 V=800.0 PL=0
MOVL C01342 V=800.0 PL=0
MOVL C01343 V=800.0 PL=0
MOVL C01344 V=800.0 PL=0
MOVL C01345 V=800.0 PL=0
MOVL C01346 V=800.0 PL=0
MOVL C01347 V=800.0 PL=0
MOVL C01348 V=800.0 PL=0
MOVL C01349 V=800.0 PL=0
MOVL C01350 V=800.0 PL=0
MOVL C01351 V=800.0 PL=0
MOVL C01352 V=800.0 PL=0
MOVL C01353 V=800.0 PL=0
MOVL C01354 V=800.0 PL=0
MOVL C01355 V=800.0 PL=0
MOVL C01356 V=800.0 PL=0
MOVL C01357 V=800.0 PL=0
MOVL C01358 V=800.0 PL=0
MOVL C01359 V=800.0 PL=0
MOVL C01360 V=800.0 PL=0
MOVL C01361 V=800.0 PL=0
MOVL C01362 V=800.0 PL=0
MOVL C01363 V=800.0 PL=0
MOVL C01364 V=800.0 PL=0
MOVL C01365 V=800.0 PL=0
MOVL C01366 V=800.0 PL=0
MOVL C01367 V=800.0 PL=0
MOVL C01368 V=800.0 PL=0
MOVL C01369 V=800.0 PL=0
MOVL C01370 V=800.0 PL=0
MOVL C01371 V=800.0 PL=0
MOVL C01372 V=800.0 PL=0
MOVL C01373 V=800.0 PL=0
MOVL C01374 V=800.0 PL=0
MOVL C01375 V=800.0 PL=0
MOVL C01376 V=800.0 PL=0
MOVL C01377 V=800.0 PL=0
MOVL C01378 V=800.0 PL=0
MOVL C01379 V=800.0 PL=0
MOVL C01380 V=800.0 PL=0
MOVL C01381 V=800.0 PL=0
MOVL C01382 V=800.0 PL=0
MOVL C01383 V=800.0 PL=0
MOVL C01384 V=800.0 PL=0
MOVL C01385 V=800.0 PL=0
MOVL C01386 V=800.0 PL=0
MOVL C01387 V=800.0 PL=0
MOVL C01388 V=800.0 PL=0
MOVL C01389 V=800.0 PL=0
MOVL C01390 V=800.0 PL=0
MOVL C01391 V=800.0 PL=0
MOVL C01392 V=800.0 PL=0
MOVL C01393 V=800.0 PL=0
MOVL C01394 V=800.0 PL=0
MOVL C01395 V=800.0 PL=0
MOVL C01396 V=800.0 PL=0
MOVL C01397 V=800.0 PL=0
MOVL C01398 V=800.0 PL=0
MOVL C01399 V=800.0 PL=0
MOVL C01400 V=800.0 PL=0
MOVL C01401 V=800.0 PL=0
MOVL C01402 V=800.0 PL=0
MOVL C01403 V=800.0 PL=0
MOVL C01404 V=800.0 PL=0
MOVL C01405 V=800.0 PL=0
MOVL C01406 V=800.0 PL=0
MOVL C01407 V=800.0 PL=0
MOVL C01408 V=800.0 PL=0
MOVL C01409 V=800.0 PL=0
MOVL C01410 V=800.0 PL=0
MOVL C01411 V=800.0 PL=0
MOVL C01412 V=800.0 PL=0
MOVL C01413 V=800.0 PL=0
MOVL C01414 V=800.0 PL=0
MOVL C01415 V=800.0 PL=0
MOVL C01416 V=800.0 PL=0
MOVL C01417 V=800.0 PL=0
MOVL C01418 V=800.0 PL=0
MOVL C01419 V=800.0 PL=0
MOVL C01420 V=800.0 PL=0
MOVL C01421 V=800.0 PL=0
MOVL C01422 V=800.0 PL=0
MOVL C01423 V=800.0 PL=0
MOVL C01424 V=800.0 PL=0
MOVL C01425 V=800.0 PL=0
MOVL C01426 V=800.0 PL=0
MOVL C01427 V=800.0 PL=0
MOVL C01428 V=800.0 PL=0
MOVL C01429 V=800.0 PL=0
MOVL C01430 V=800.0 PL=0
MOVL C01431 V=800.0 PL=0
MOVL C01432 V=800.0 PL=0
MOVL C01433 V=800.0 PL=0
MOVL C01434 V=800.0 PL=0
MOVL C01435 V=800.0 PL=0
MOVL C01436 V=800.0 PL=0
MOVL C01437 V=800.0 PL=0
MOVL C01438 V=800.0 PL=0
MOVL C01439 V=800.0 PL=0
MOVL C01440 V=800.0 PL=0
MOVL C01441 V=800.0 PL=0
MOVL C01442 V=800.0 PL=0
MOVL C01443 V=800.0 PL=0
MOVL C01444 V=800.0 PL=0
MOVL C01445 V=800.0 PL=0
MOVL C01446 V=800.0 PL=0
MOVL C01447 V=800.0 PL=0
MOVL C01448 V=800.0 PL=0
MOVL C01449 V=800.0 PL=0
MOVL C01450 V=800.0 PL=0
MOVL C01451 V=800.0 PL=0
MOVL C01452 V=800.0 PL=0
MOVL C01453 V=800.0 PL=0
MOVL C01454 V=800.0 PL=0
MOVL C01455 V=800.0 PL=0
MOVL C01456 V=800.0 PL=0
MOVL C01457 V=800.0 PL=0
MOVL C01458 V=800.0 PL=0
MOVL C01459 V=800.0 PL=0
MOVL C01460 V=800.0 PL=0
MOVL C01461 V=800.0 PL=0
MOVL C01462 V=800.0 PL=0
MOVL C01463 V=800.0 PL=0
MOVL C01464 V=800.0 PL=0
MOVL C01465 V=800.0 PL=0
MOVL C01466 V=800.0 PL=0
MOVL C01467 V=800.0 PL=0
MOVL C01468 V=800.0 PL=0
MOVL C01469 V=800.0 PL=0
MOVL C01470 V=800.0 PL=0
MOVL C01471 V=800.0 PL=0
MOVL C01472 V=800.0 PL=0
MOVL C01473 V=800.0 PL=0
MOVL C01474 V=800.0 PL=0
MOVL C01475 V=800.0 PL=0
MOVL C01476 V=800.0 PL=0
MOVL C01477 V=800.0 PL=0
MOVL C01478 V=800.0 PL=0
MOVL C01479 V=800.0 PL=0
MOVL C01480 V=800.0 PL=0
MOVL C01481 V=800.0 PL=0
MOVL C01482 V=800.0 PL=0
MOVL C01483 V=800.0 PL=0
MOVL C01484 V=800.0 PL=0
MOVL C01485 V=800.0 PL=0
MOVL C01486 V=800.0 PL=0
MOVL C01487 V=800.0 PL=0
MOVL C01488 V=800.0 PL=0
MOVL C01489 V=800.0 PL=0
MOVL C01490 V=800.0 PL=0
MOVL C01491 V=800.0 PL=0
MOVL C01492 V=800.0 PL=0
MOVL C01493 V=800.0 PL=0
MOVL C01494 V=800.0 PL=0
MOVL C01495 V=800.0 PL=0
MOVL C01496 V=800.0 PL=0
MOVL C01497 V=800.0 PL=0
MOVL C01498 V=800.0 PL=0
MOVL C01499 V=800.0 PL=0
MOVL C01500 V=800.0 PL=0
MOVL C01501 V=800.0 PL=0
MOVL C01502 V=800.0 PL=0
MOVL C01503 V=800.0 PL=0
MOVL C01504 V=800.0 PL=0
MOVL C01505 V=800.0 PL=0
MOVL C01506 V=800.0 PL=0
MOVL C01507 V=800.0 PL=0
MOVL C01508 V=800.0 PL=0
MOVL C01509 V=800.0 PL=0
MOVL C01510 V=800.0 PL=0
MOVL C01511 V=800.0 PL=0
MOVL C01512 V=800.0 PL=0
MOVL C01513 V=800.0 PL=0
MOVL C01514 V=800.0 PL=0
MOVL C01515 V=800.0 PL=0
MOVL C01516 V=800.0 PL=0
MOVL C01517 V=800.0 PL=0
MOVL C01518 V=800.0 PL=0
MOVL C01519 V=800.0 PL=0
MOVL C01520 V=800.0 PL=0
MOVL C01521 V=800.0 PL=0
MOVL C01522 V=800.0 PL=0
MOVL C01523 V=800.0 PL=0
MOVL C01524 V=800.0 PL=0
MOVL C01525 V=800.0 PL=0
MOVL C01526 V=800.0 PL=0
MOVL C01527 V=800.0 PL=0
MOVL C01528 V=800.0 PL=0
MOVL C01529 V=800.0 PL=0
MOVL C01530 V=800.0 PL=0
MOVL C01531 V=800.0 PL=0
MOVL C01532 V=800.0 PL=0
MOVL C01533 V=800.0 PL=0
MOVL C01534 V=800.0 PL=0
MOVL C01535 V=800.0 PL=0
MOVL C01536 V=800.0 PL=0
MOVL C01537 V=800.0 PL=0
MOVL C01538 V=800.0 PL=0
MOVL C01539 V=800.0 PL=0
MOVL C01540 V=800.0 PL=0
MOVL C01541 V=800.0 PL=0
MOVL C01542 V=800.0 PL=0
MOVL C01543 V=800.0 PL=0
MOVL C01544 V=800.0 PL=0
MOVL C01545 V=800.0 PL=0
MOVL C01546 V=800.0 PL=0
MOVL C01547 V=800.0 PL=0
MOVL C01548 V=800.0 PL=0
MOVL C01549 V=800.0 PL=0
MOVL C01550 V=800.0 PL=0
MOVL C01551 V=800.0 PL=0
MOVL C01552 V=800.0 PL=0
MOVL C01553 V=800.0 PL=0
MOVL C01554 V=800.0 PL=0
MOVL C01555 V=800.0 PL=0
MOVL C01556 V=800.0 PL=0
MOVL C01557 V=800.0 PL=0
MOVL C01558 V=800.0 PL=0
MOVL C01559 V=800.0 PL=0
MOVL C01560 V=800.0 PL=0
MOVL C01561 V=800.0 PL=0
MOVL C01562 V=800.0 PL=0
MOVL C01563 V=800.0 PL=0
MOVL C01564 V=800.0 PL=0
MOVL C01565 V=800.0 PL=0
MOVL C01566 V=800.0 PL=0
MOVL C01567 V=800.0 PL=0
MOVL C01568 V=800.0 PL=0
MOVL C01569 V=800.0 PL=0
MOVL C01570 V=800.0 PL=0
MOVL C01571 V=800.0 PL=0
MOVL C01572 V=800.0 PL=0
MOVL C01573 V=800.0 PL=0
MOVL C01574 V=800.0 PL=0
MOVL C01575 V=800.0 PL=0
MOVL C01576 V=800.0 PL=0
MOVL C01577 V=800.0 PL=0
MOVL C01578 V=800.0 PL=0
MOVL C01579 V=800.0 PL=0
MOVL C01580 V=800.0 PL=0
MOVL C01581 V=800.0 PL=0
MOVL C01582 V=800.0 PL=0
MOVL C01583 V=800.0 PL=0
MOVL C01584 V=800.0 PL=0
MOVL C01585 V=800.0 PL=0
MOVL C01586 V=800.0 PL=0
MOVL C01587 V=800.0 PL=0
MOVL C01588 V=800.0 PL=0
MOVL C01589 V=800.0 PL=0
MOVL C01590 V=800.0 PL=0
MOVL C01591 V=800.0 PL=0
MOVL C01592 V=800.0 PL=0
MOVL C01593 V=800.0 PL=0
MOVL C01594 V=800.0 PL=0
MOVL C01595 V=800.0 PL=0
MOVL C01596 V=800.0 PL=0
MOVL C01597 V=800.0 PL=0
MOVL C01598 V=800.0 PL=0
MOVL C01599 V=800.0 PL=0
MOVL C01600 V=800.0 PL=0
MOVL C01601 V=800.0 PL=0
MOVL C01602 V=800.0 PL=0
MOVL C01603 V=800.0 PL=0
MOVL C01604 V=800.0 PL=0
MOVL C01605 V=800.0 PL=0
MOVL C01606 V=800.0 PL=0
MOVL C01607 V=800.0 PL=0
MOVL C01608 V=800.0 PL=0
MOVL C01609 V=800.0 PL=0
MOVL C01610 V=800.0 PL=0
MOVL C01611 V=800.0 PL=0
MOVL C01612 V=800.0 PL=0
MOVL C01613 V=800.0 PL=0
MOVL C01614 V=800.0 PL=0
MOVL C01615 V=800.0 PL=0
MOVL C01616 V=800.0 PL=0
MOVL C01617 V=800.0 PL=0
MOVL C01618 V=800.0 PL=0
MOVL C01619 V=800.0 PL=0
MOVL C01620 V=800.0 PL=0
MOVL C01621 V=800.0 PL=0
MOVL C01622 V=800.0 PL=0
MOVL C01623 V=800.0 PL=0
MOVL C01624 V=800.0 PL=0
MOVL C01625 V=800.0 PL=0
MOVL C01626 V=800.0 PL=0
MOVL C01627 V=800.0 PL=0
MOVL C01628 V=800.0 PL=0
MOVL C01629 V=800.0 PL=0
MOVL C01630 V=800.0 PL=0
MOVL C01631 V=800.0 PL=0
MOVL C01632 V=800.0 PL=0
MOVL C01633 V=800.0 PL=0
MOVL C01634 V=800.0 PL=0
MOVL C01635 V=800.0 PL=0
MOVL C01636 V=800.0 PL=0
MOVL C01637 V=800.0 PL=0
MOVL C01638 V=800.0 PL=0
MOVL C01639 V=800.0 PL=0
MOVL C01640 V=800.0 PL=0
MOVL C01641 V=800.0 PL=0
MOVL C01642 V=800.0 PL=0
MOVL C01643 V=800.0 PL=0
MOVL C01644 V=800.0 PL=0
MOVL C01645 V=800.0 PL=0
MOVL C01646 V=800.0 PL=0
MOVL C01647 V=800.0 PL=0
MOVL C01648 V=800.0 PL=0
MOVL C01649 V=800.0 PL=0
MOVL C01650 V=800.0 PL=0
MOVL C01651 V=800.0 PL=0
MOVL C01652 V=800.0 PL=0
MOVL C01653 V=800.0 PL=0
MOVL C01654 V=800.0 PL=0
MOVL C01655 V=800.0 PL=0
MOVL C01656 V=800.0 PL=0
MOVL C01657 V=800.0 PL=0
MOVL C01658 V=800.0 PL=0
MOVL C01659 V=800.0 PL=0
MOVL C01660 V=800.0 PL=0
MOVL C01661 V=800.0 PL=0
MOVL C01662 V=800.0 PL=0
MOVL C01663 V=800.0 PL=0
MOVL C01664 V=800.0 PL=0
MOVL C01665 V=800.0 PL=0
MOVL C01666 V=800.0 PL=0
MOVL C01667 V=800.0 PL=0
MOVL C01668 V=800.0 PL=0
MOVL C01669 V=800.0 PL=0
MOVL C01670 V=800.0 PL=0
MOVL C01671 V=800.0 PL=0
MOVL C01672 V=800.0 PL=0
MOVL C01673 V=800.0 PL=0
MOVL C01674 V=800.0 PL=0
MOVL C01675 V=800.0 PL=0
MOVL C01676 V=800.0 PL=0
MOVL C01677 V=800.0 PL=0
MOVL C01678 V=800.0 PL=0
MOVL C01679 V=800.0 PL=0
MOVL C01680 V=800.0 PL=0
MOVL C01681 V=800.0 PL=0
MOVL C01682 V=800.0 PL=0
MOVL C01683 V=800.0 PL=0
MOVL C01684 V=800.0 PL=0
MOVL C01685 V=800.0 PL=0
MOVL C01686 V=800.0 PL=0
MOVL C01687 V=800.0 PL=0
MOVL C01688 V=800.0 PL=0
MOVL C01689 V=800.0 PL=0
MOVL C01690 V=800.0 PL=0
MOVL C01691 V=800.0 PL=0
MOVL C01692 V=800.0 PL=0
MOVL C01693 V=800.0 PL=0
MOVL C01694 V=800.0 PL=0
MOVL C01695 V=800.0 PL=0
MOVL C01696 V=800.0 PL=0
MOVL C01697 V=800.0 PL=0
MOVL C01698 V=800.0 PL=0
MOVL C01699 V=800.0 PL=0
MOVL C01700 V=800.0 PL=0
MOVL C01701 V=800.0 PL=0
MOVL C01702 V=800.0 PL=0
MOVL C01703 V=800.0 PL=0
MOVL C01704 V=800.0 PL=0
MOVL C01705 V=800.0 PL=0
MOVL C01706 V=800.0 PL=0
MOVL C01707 V=800.0 PL=0
MOVL C01708 V=800.0 PL=0
MOVL C01709 V=800.0 PL=0
MOVL C01710 V=800.0 PL=0
MOVL C01711 V=800.0 PL=0
MOVL C01712 V=800.0 PL=0
MOVL C01713 V=800.0 PL=0
MOVL C01714 V=800.0 PL=0
MOVL C01715 V=800.0 PL=0
MOVL C01716 V=800.0 PL=0
MOVL C01717 V=800.0 PL=0
MOVL C01718 V=800.0 PL=0
MOVL C01719 V=800.0 PL=0
MOVL C01720 V=800.0 PL=0
MOVL C01721 V=800.0 PL=0
MOVL C01722 V=800.0 PL=0
MOVL C01723 V=800.0 PL=0
MOVL C01724 V=800.0 PL=0
MOVL C01725 V=800.0 PL=0
MOVL C01726 V=800.0 PL=0
MOVL C01727 V=800.0 PL=0
MOVL C01728 V=800.0 PL=0
MOVL C01729 V=800.0 PL=0
MOVL C01730 V=800.0 PL=0
MOVL C01731 V=800.0 PL=0
MOVL C01732 V=800.0 PL=0
MOVL C01733 V=800.0 PL=0
MOVL C01734 V=800.0 PL=0
MOVL C01735 V=800.0 PL=0
MOVL C01736 V=800.0 PL=0
MOVL C01737 V=800.0 PL=0
MOVL C01738 V=800.0 PL=0
MOVL C01739 V=800.0 PL=0
MOVL C01740 V=800.0 PL=0
MOVL C01741 V=800.0 PL=0
MOVL C01742 V=800.0 PL=0
MOVL C01743 V=800.0 PL=0
MOVL C01744 V=800.0 PL=0
MOVL C01745 V=800.0 PL=0
MOVL C01746 V=800.0 PL=0
MOVL C01747 V=800.0 PL=0
MOVL C01748 V=800.0 PL=0
MOVL C01749 V=800.0 PL=0
MOVL C01750 V=800.0 PL=0
MOVL C01751 V=800.0 PL=0
MOVL C01752 V=800.0 PL=0
MOVL C01753 V=800.0 PL=0
MOVL C01754 V=800.0 PL=0
MOVL C01755 V=800.0 PL=0
MOVL C01756 V=800.0 PL=0
MOVL C01757 V=800.0 PL=0
MOVL C01758 V=800.0 PL=0
MOVL C01759 V=800.0 PL=0
MOVL C01760 V=800.0 PL=0
MOVL C01761 V=800.0 PL=0
MOVL C01762 V=800.0 PL=0
MOVL C01763 V=800.0 PL=0
MOVL C01764 V=800.0 PL=0
MOVL C01765 V=800.0 PL=0
MOVL C01766 V=800.0 PL=0
MOVL C01767 V=800.0 PL=0
MOVL C01768 V=800.0 PL=0
MOVL C01769 V=800.0 PL=0
MOVL C01770 V=800.0 PL=0
MOVL C01771 V=800.0 PL=0
MOVL C01772 V=800.0 PL=0
MOVL C01773 V=800.0 PL=0
MOVL C01774 V=800.0 PL=0
MOVL C01775 V=800.0 PL=0
MOVL C01776 V=800.0 PL=0
MOVL C01777 V=800.0 PL=0
MOVL C01778 V=800.0 PL=0
MOVL C01779 V=800.0 PL=0
MOVL C01780 V=800.0 PL=0
MOVL C01781 V=800.0 PL=0
MOVL C01782 V=800.0 PL=0
MOVL C01783 V=800.0 PL=0
MOVL C01784 V=800.0 PL=0
MOVL C01785 V=800.0 PL=0
MOVL C01786 V=800.0 PL=0
MOVL C01787 V=800.0 PL=0
MOVL C01788 V=800.0 PL=0
MOVL C01789 V=800.0 PL=0
MOVL C01790 V=800.0 PL=0
MOVL C01791 V=800.0 PL=0
MOVL C01792 V=800.0 PL=0
MOVL C01793 V=800.0 PL=0
MOVL C01794 V=800.0 PL=0
MOVL C01795 V=800.0 PL=0
MOVL C01796 V=800.0 PL=0
MOVL C01797 V=800.0 PL=0
MOVL C01798 V=800.0 PL=0
MOVL C01799 V=800.0 PL=0
MOVL C01800 V=800.0 PL=0
MOVL C01801 V=800.0 PL=0
MOVL C01802 V=800.0 PL=0
MOVL C01803 V=800.0 PL=0
MOVL C01804 V=800.0 PL=0
MOVL C01805 V=800.0 PL=0
MOVL C01806 V=800.0 PL=0
MOVL C01807 V=800.0 PL=0
MOVL C01808 V=800.0 PL=0
MOVL C01809 V=800.0 PL=0
MOVL C01810 V=800.0 PL=0
MOVL C01811 V=800.0 PL=0
MOVL C01812 V=800.0 PL=0
MOVL C01813 V=800.0 PL=0
MOVL C01814 V=800.0 PL=0
MOVL C01815 V=800.0 PL=0
MOVL C01816 V=800.0 PL=0
MOVL C01817 V=800.0 PL=0
MOVL C01818 V=800.0 PL=0
MOVL C01819 V=800.0 PL=0
MOVL C01820 V=800.0 PL=0
MOVL C01821 V=800.0 PL=0
MOVL C01822 V=800.0 PL=0
MOVL C01823 V=800.0 PL=0
MOVL C01824 V=800.0 PL=0
MOVL C01825 V=800.0 PL=0
MOVL C01826 V=800.0 PL=0
MOVL C01827 V=800.0 PL=0
MOVL C01828 V=800.0 PL=0
MOVL C01829 V=800.0 PL=0
MOVL C01830 V=800.0 PL=0
MOVL C01831 V=800.0 PL=0
MOVL C01832 V=800.0 PL=0
MOVL C01833 V=800.0 PL=0
MOVL C01834 V=800.0 PL=0
MOVL C01835 V=800.0 PL=0
MOVL C01836 V=800.0 PL=0
MOVL C01837 V=800.0 PL=0
MOVL C01838 V=800.0 PL=0
MOVL C01839 V=800.0 PL=0
MOVL C01840 V=800.0 PL=0
MOVL C01841 V=800.0 PL=0
MOVL C01842 V=800.0 PL=0
MOVL C01843 V=800.0 PL=0
MOVL C01844 V=800.0 PL=0
MOVL C01845 V=800.0 PL=0
MOVL C01846 V=800.0 PL=0
MOVL C01847 V=800.0 PL=0
MOVL C01848 V=800.0 PL=0
MOVL C01849 V=800.0 PL=0
MOVL C01850 V=800.0 PL=0
MOVL C01851 V=800.0 PL=0
MOVL C01852 V=800.0 PL=0
MOVL C01853 V=800.0 PL=0
MOVL C01854 V=800.0 PL=0
MOVL C01855 V=800.0 PL=0
MOVL C01856 V=800.0 PL=0
MOVL C01857 V=800.0 PL=0
MOVL C01858 V=800.0 PL=0
MOVL C01859 V=800.0 PL=0
MOVL C01860 V=800.0 PL=0
MOVL C01861 V=800.0 PL=0
MOVL C01862 V=800.0 PL=0
MOVL C01863 V=800.0 PL=0
MOVL C01864 V=800.0 PL=0
MOVL C01865 V=800.0 PL=0
MOVL C01866 V=800.0 PL=0
MOVL C01867 V=800.0 PL=0
MOVL C01868 V=800.0 PL=0
MOVL C01869 V=800.0 PL=0
MOVL C01870 V=800.0 PL=0
MOVL C01871 V=800.0 PL=0
MOVL C01872 V=800.0 PL=0
MOVL C01873 V=800.0 PL=0
MOVL C01874 V=800.0 PL=0
MOVL C01875 V=800.0 PL=0
MOVL C01876 V=800.0 PL=0
MOVL C01877 V=800.0 PL=0
MOVL C01878 V=800.0 PL=0
MOVL C01879 V=800.0 PL=0
MOVL C01880 V=800.0 PL=0
MOVL C01881 V=800.0 PL=0
MOVL C01882 V=800.0 PL=0
MOVL C01883 V=800.0 PL=0
MOVL C01884 V=800.0 PL=0
MOVL C01885 V=800.0 PL=0
MOVL C01886 V=800.0 PL=0
MOVL C01887 V=800.0 PL=0
MOVL C01888 V=800.0 PL=0
MOVL C01889 V=800.0 PL=0
MOVL C01890 V=800.0 PL=0
MOVL C01891 V=800.0 PL=0
MOVL C01892 V=800.0 PL=0
MOVL C01893 V=800.0 PL=0
MOVL C01894 V=800.0 PL=0
MOVL C01895 V=800.0 PL=0
MOVL C01896 V=800.0 PL=0
MOVL C01897 V=800.0 PL=0
MOVL C01898 V=800.0 PL=0
MOVL C01899 V=800.0 PL=0
MOVL C01900 V=800.0 PL=0
MOVL C01901 V=800.0 PL=0
MOVL C01902 V=800.0 PL=0
MOVL C01903 V=800.0 PL=0
MOVL C01904 V=800.0 PL=0
MOVL C01905 V=800.0 PL=0
MOVL C01906 V=800.0 PL=0
MOVL C01907 V=800.0 PL=0
MOVL C01908 V=800.0 PL=0
MOVL C01909 V=800.0 PL=0
MOVL C01910 V=800.0 PL=0
MOVL C01911 V=800.0 PL=0
MOVL C01912 V=800.0 PL=0
MOVL C01913 V=800.0 PL=0
MOVL C01914 V=800.0 PL=0
MOVL C01915 V=800.0 PL=0
MOVL C01916 V=800.0 PL=0
MOVL C01917 V=800.0 PL=0
MOVL C01918 V=800.0 PL=0
MOVL C01919 V=800.0 PL=0
MOVL C01920 V=800.0 PL=0
MOVL C01921 V=800.0 PL=0
MOVL C01922 V=800.0 PL=0
MOVL C01923 V=800.0 PL=0
MOVL C01924 V=800.0 PL=0
MOVL C01925 V=800.0 PL=0
MOVL C01926 V=800.0 PL=0
MOVL C01927 V=800.0 PL=0
MOVL C01928 V=800.0 PL=0
MOVL C01929 V=800.0 PL=0
MOVL C01930 V=800.0 PL=0
MOVL C01931 V=800.0 PL=0
MOVL C01932 V=800.0 PL=0
MOVL C01933 V=800.0 PL=0
MOVL C01934 V=800.0 PL=0
MOVL C01935 V=800.0 PL=0
MOVL C01936 V=800.0 PL=0
MOVL C01937 V=800.0 PL=0
MOVL C01938 V=800.0 PL=0
MOVL C01939 V=800.0 PL=0
MOVL C01940 V=800.0 PL=0
MOVL C01941 V=800.0 PL=0
MOVL C01942 V=800.0 PL=0
MOVL C01943 V=800.0 PL=0
MOVL C01944 V=800.0 PL=0
MOVL C01945 V=800.0 PL=0
MOVL C01946 V=800.0 PL=0
MOVL C01947 V=800.0 PL=0
MOVL C01948 V=800.0 PL=0
MOVL C01949 V=800.0 PL=0
MOVL C01950 V=800.0 PL=0
MOVL C01951 V=800.0 PL=0
MOVL C01952 V=800.0 PL=0
MOVL C01953 V=800.0 PL=0
MOVL C01954 V=800.0 PL=0
MOVL C01955 V=800.0 PL=0
MOVL C01956 V=800.0 PL=0
MOVL C01957 V=800.0 PL=0
MOVL C01958 V=800.0 PL=0
MOVL C01959 V=800.0 PL=0
MOVL C01960 V=800.0 PL=0
MOVL C01961 V=800.0 PL=0
MOVL C01962 V=800.0 PL=0
MOVL C01963 V=800.0 PL=0
MOVL C01964 V=800.0 PL=0
MOVL C01965 V=800.0 PL=0
MOVL C01966 V=800.0 PL=0
MOVL C01967 V=800.0 PL=0
MOVL C01968 V=800.0 PL=0
MOVL C01969 V=800.0 PL=0
MOVL C01970 V=800.0 PL=0
MOVL C01971 V=800.0 PL=0
MOVL C01972 V=800.0 PL=0
MOVL C01973 V=800.0 PL=0
MOVL C01974 V=800.0 PL=0
MOVL C01975 V=800.0 PL=0
MOVL C01976 V=800.0 PL=0
MOVL C01977 V=800.0 PL=0
MOVL C01978 V=800.0 PL=0
MOVL C01979 V=800.0 PL=0
MOVL C01980 V=800.0 PL=0
MOVL C01981 V=800.0 PL=0
MOVL C01982 V=800.0 PL=0
MOVL C01983 V=800.0 PL=0
MOVL C01984 V=800.0 PL=0
MOVL C01985 V=800.0 PL=0
MOVL C01986 V=800.0 PL=0
MOVL C01987 V=800.0 PL=0
MOVL C01988 V=800.0 PL=0
MOVL C01989 V=800.0 PL=0
MOVL C01990 V=800.0 PL=0
MOVL C01991 V=800.0 PL=0
MOVL C01992 V=800.0 PL=0
MOVL C01993 V=800.0 PL=0
MOVL C01994 V=800.0 PL=0
MOVL C01995 V=800.0 PL=0
MOVL C01996 V=800.0 PL=0
MOVL C01997 V=800.0 PL=0
MOVL C01998 V=800.0 PL=0
MOVL C01999 V=800.0 PL=0
MOVL C02000 V=800.0 PL=0
MOVL C02001 V=800.0 PL=0
MOVL C02002 V=800.0 PL=0
MOVL C02003 V=800.0 PL=0
MOVL C02004 V=800.0 PL=0
MOVL C02005 V=800.0 PL=0
MOVL C02006 V=800.0 PL=0
MOVL C02007 V=800.0 PL=0
MOVL C02008 V=800.0 PL=0
MOVL C02009 V=800.0 PL=0
MOVL C02010 V=800.0 PL=0
MOVL C02011 V=800.0 PL=0
MOVL C02012 V=800.0 PL=0
MOVL C02013 V=800.0 PL=0
MOVL C02014 V=800.0 PL=0
MOVL C02015 V=800.0 PL=0
MOVL C02016 V=800.0 PL=0
MOVL C02017 V=800.0 PL=0
MOVL C02018 V=800.0 PL=0
MOVL C02019 V=800.0 PL=0
MOVL C02020 V=800.0 PL=0
MOVL C02021 V=800.0 PL=0
MOVL C02022 V=800.0 PL=0
MOVL C02023 V=800.0 PL=0
MOVL C02024 V=800.0 PL=0
MOVL C02025 V=800.0 PL=0
MOVL C02026 V=800.0 PL=0
MOVL C02027 V=800.0 PL=0
MOVL C02028 V=800.0 PL=0
MOVL C02029 V=800.0 PL=0
MOVL C02030 V=800.0 PL=0
MOVL C02031 V=800.0 PL=0
MOVL C02032 V=800.0 PL=0
MOVL C02033 V=800.0 PL=0
MOVL C02034 V=800.0 PL=0
MOVL C02035 V=800.0 PL=0
MOVL C02036 V=800.0 PL=0
MOVL C02037 V=800.0 PL=0
MOVL C02038 V=800.0 PL=0
MOVL C02039 V=800.0 PL=0
MOVL C02040 V=800.0 PL=0
MOVL C02041 V=800.0 PL=0
MOVL C02042 V=800.0 PL=0
MOVL C02043 V=800.0 PL=0
MOVL C02044 V=800.0 PL=0
MOVL C02045 V=800.0 PL=0
MOVL C02046 V=800.0 PL=0
MOVL C02047 V=800.0 PL=0
MOVL C02048 V=800.0 PL=0
MOVL C02049 V=800.0 PL=0
MOVL C02050 V=800.0 PL=0
MOVL C02051 V=800.0 PL=0
MOVL C02052 V=800.0 PL=0
MOVL C02053 V=800.0 PL=0
MOVL C02054 V=800.0 PL=0
MOVL C02055 V=800.0 PL=0
MOVL C02056 V=800.0 PL=0
MOVL C02057 V=800.0 PL=0
MOVL C02058 V=800.0 PL=0
MOVL C02059 V=800.0 PL=0
MOVL C02060 V=800.0 PL=0
MOVL C02061 V=800.0 PL=0
MOVL C02062 V=800.0 PL=0
MOVL C02063 V=800.0 PL=0
MOVL C02064 V=800.0 PL=0
MOVL C02065 V=800.0 PL=0
MOVL C02066 V=800.0 PL=0
MOVL C02067 V=800.0 PL=0
MOVL C02068 V=800.0 PL=0
MOVL C02069 V=800.0 PL=0
MOVL C02070 V=800.0 PL=0
MOVL C02071 V=800.0 PL=0
MOVL C02072 V=800.0 PL=0
MOVL C02073 V=800.0 PL=0
MOVL C02074 V=800.0 PL=0
MOVL C02075 V=800.0 PL=0
MOVL C02076 V=800.0 PL=0
MOVL C02077 V=800.0 PL=0
MOVL C02078 V=800.0 PL=0
MOVL C02079 V=800.0 PL=0
MOVL C02080 V=800.0 PL=0
MOVL C02081 V=800.0 PL=0
MOVL C02082 V=800.0 PL=0
MOVL C02083 V=800.0 PL=0
MOVL C02084 V=800.0 PL=0
MOVL C02085 V=800.0 PL=0
MOVL C02086 V=800.0 PL=0
MOVL C02087 V=800.0 PL=0
MOVL C02088 V=800.0 PL=0
MOVL C02089 V=800.0 PL=0
MOVL C02090 V=800.0 PL=0
MOVL C02091 V=800.0 PL=0
MOVL C02092 V=800.0 PL=0
MOVL C02093 V=800.0 PL=0
MOVL C02094 V=800.0 PL=0
MOVL C02095 V=800.0 PL=0
MOVL C02096 V=800.0 PL=0
MOVL C02097 V=800.0 PL=0
MOVL C02098 V=800.0 PL=0
MOVL C02099 V=800.0 PL=0
MOVL C02100 V=800.0 PL=0
MOVL C02101 V=800.0 PL=0
MOVL C02102 V=800.0 PL=0
MOVL C02103 V=800.0 PL=0
MOVL C02104 V=800.0 PL=0
MOVL C02105 V=800.0 PL=0
MOVL C02106 V=800.0 PL=0
MOVL C02107 V=800.0 PL=0
MOVL C02108 V=800.0 PL=0
MOVL C02109 V=800.0 PL=0
MOVL C02110 V=800.0 PL=0
MOVL C02111 V=800.0 PL=0
MOVL C02112 V=800.0 PL=0
MOVL C02113 V=800.0 PL=0
MOVL C02114 V=800.0 PL=0
MOVL C02115 V=800.0 PL=0
MOVL C02116 V=800.0 PL=0
MOVL C02117 V=800.0 PL=0
MOVL C02118 V=800.0 PL=0
MOVL C02119 V=800.0 PL=0
MOVL C02120 V=800.0 PL=0
MOVL C02121 V=800.0 PL=0
MOVL C02122 V=800.0 PL=0
MOVL C02123 V=800.0 PL=0
MOVL C02124 V=800.0 PL=0
MOVL C02125 V=800.0 PL=0
MOVL C02126 V=800.0 PL=0
MOVL C02127 V=800.0 PL=0
MOVL C02128 V=800.0 PL=0
MOVL C02129 V=800.0 PL=0
MOVL C02130 V=800.0 PL=0
MOVL C02131 V=800.0 PL=0
MOVL C02132 V=800.0 PL=0
MOVL C02133 V=800.0 PL=0
MOVL C02134 V=800.0 PL=0
MOVL C02135 V=800.0 PL=0
MOVL C02136 V=800.0 PL=0
MOVL C02137 V=800.0 PL=0
MOVL C02138 V=800.0 PL=0
MOVL C02139 V=800.0 PL=0
MOVL C02140 V=800.0 PL=0
MOVL C02141 V=800.0 PL=0
MOVL C02142 V=800.0 PL=0
MOVL C02143 V=800.0 PL=0
MOVL C02144 V=800.0 PL=0
MOVL C02145 V=800.0 PL=0
MOVL C02146 V=800.0 PL=0
MOVL C02147 V=800.0 PL=0
MOVL C02148 V=800.0 PL=0
MOVL C02149 V=800.0 PL=0
MOVL C02150 V=800.0 PL=0
MOVL C02151 V=800.0 PL=0
MOVL C02152 V=800.0 PL=0
MOVL C02153 V=800.0 PL=0
MOVL C02154 V=800.0 PL=0
MOVL C02155 V=800.0 PL=0
MOVL C02156 V=800.0 PL=0
MOVL C02157 V=800.0 PL=0
MOVL C02158 V=800.0 PL=0
MOVL C02159 V=800.0 PL=0
MOVL C02160 V=800.0 PL=0
MOVL C02161 V=800.0 PL=0
MOVL C02162 V=800.0 PL=0
MOVL C02163 V=800.0 PL=0
MOVL C02164 V=800.0 PL=0
MOVL C02165 V=800.0 PL=0
MOVL C02166 V=800.0 PL=0
MOVL C02167 V=800.0 PL=0
MOVL C02168 V=800.0 PL=0
MOVL C02169 V=800.0 PL=0
MOVL C02170 V=800.0 PL=0
MOVL C02171 V=800.0 PL=0
MOVL C02172 V=800.0 PL=0
MOVL C02173 V=800.0 PL=0
MOVL C02174 V=800.0 PL=0
MOVL C02175 V=800.0 PL=0
MOVL C02176 V=800.0 PL=0
MOVL C02177 V=800.0 PL=0
MOVL C02178 V=800.0 PL=0
MOVL C02179 V=800.0 PL=0
MOVL C02180 V=800.0 PL=0
MOVL C02181 V=800.0 PL=0
MOVL C02182 V=800.0 PL=0
MOVL C02183 V=800.0 PL=0
MOVL C02184 V=800.0 PL=0
MOVL C02185 V=800.0 PL=0
MOVL C02186 V=800.0 PL=0
MOVL C02187 V=800.0 PL=0
MOVL C02188 V=800.0 PL=0
MOVL C02189 V=800.0 PL=0
MOVL C02190 V=800.0 PL=0
MOVL C02191 V=800.0 PL=0
MOVL C02192 V=800.0 PL=0
MOVL C02193 V=800.0 PL=0
MOVL C02194 V=800.0 PL=0
MOVL C02195 V=800.0 PL=0
MOVL C02196 V=800.0 PL=0
MOVL C02197 V=800.0 PL=0
MOVL C02198 V=800.0 PL=0
MOVL C02199 V=800.0 PL=0
MOVL C02200 V=800.0 PL=0
MOVL C02201 V=800.0 PL=0
MOVL C02202 V=800.0 PL=0
MOVL C02203 V=800.0 PL=0
MOVL C02204 V=800.0 PL=0
MOVL C02205 V=800.0 PL=0
MOVL C02206 V=800.0 PL=0
MOVL C02207 V=800.0 PL=0
MOVL C02208 V=800.0 PL=0
MOVL C02209 V=800.0 PL=0
MOVL C02210 V=800.0 PL=0
MOVL C02211 V=800.0 PL=0
MOVL C02212 V=800.0 PL=0
MOVL C02213 V=800.0 PL=0
MOVL C02214 V=800.0 PL=0
MOVL C02215 V=800.0 PL=0
MOVL C02216 V=800.0 PL=0
MOVL C02217 V=800.0 PL=0
MOVL C02218 V=800.0 PL=0
MOVL C02219 V=800.0 PL=0
MOVL C02220 V=800.0 PL=0
MOVL C02221 V=800.0 PL=0
MOVL C02222 V=800.0 PL=0
MOVL C02223 V=800.0 PL=0
MOVL C02224 V=800.0 PL=0
MOVL C02225 V=800.0 PL=0
MOVL C02226 V=800.0 PL=0
MOVL C02227 V=800.0 PL=0
MOVL C02228 V=800.0 PL=0
MOVL C02229 V=800.0 PL=0
MOVL C02230 V=800.0 PL=0
MOVL C02231 V=800.0 PL=0
MOVL C02232 V=800.0 PL=0
MOVL C02233 V=800.0 PL=0
MOVL C02234 V=800.0 PL=0
MOVL C02235 V=800.0 PL=0
MOVL C02236 V=800.0 PL=0
MOVL C02237 V=800.0 PL=0
MOVL C02238 V=800.0 PL=0
MOVL C02239 V=800.0 PL=0
MOVL C02240 V=800.0 PL=0
MOVL C02241 V=800.0 PL=0
MOVL C02242 V=800.0 PL=0
MOVL C02243 V=800.0 PL=0
MOVL C02244 V=800.0 PL=0
MOVL C02245 V=800.0 PL=0
MOVL C02246 V=800.0 PL=0
MOVL C02247 V=800.0 PL=0
MOVL C02248 V=800.0 PL=0
MOVL C02249 V=800.0 PL=0
MOVL C02250 V=800.0 PL=0
MOVL C02251 V=800.0 PL=0
MOVL C02252 V=800.0 PL=0
MOVL C02253 V=800.0 PL=0
MOVL C02254 V=800.0 PL=0
MOVL C02255 V=800.0 PL=0
MOVL C02256 V=800.0 PL=0
MOVL C02257 V=800.0 PL=0
MOVL C02258 V=800.0 PL=0
MOVL C02259 V=800.0 PL=0
MOVL C02260 V=800.0 PL=0
MOVL C02261 V=800.0 PL=0
MOVL C02262 V=800.0 PL=0
MOVL C02263 V=800.0 PL=0
MOVL C02264 V=800.0 PL=0
MOVL C02265 V=800.0 PL=0
